  case (it.dir) of
  DIR_DOWN:
    (* Запись родителя в стек *)
    if (n > 99) then msg:='CheckValid: Stack overflow'; {goto __error} end_if;
    stack[n] := it.item;
    n:=n+1;
  DIR_UP:
    (* Извлечение из стека *)
    if (is_poly(it.item)) then  (* элемент - родитель *)
    
      (* Выборка потомства из стека *)
      m:=0;
      while (stack[n-1]<>it.item) do
        n:=n-1;
        if (m > 15) then msg:='CheckValid: Kids overflow'; {goto __error} end_if;
        kids[m]:=stack[n];
        m:=m+1;
      end_while;
      
      (* Анализ потомства *)
      for im:=0 to m-1 do
        PIT:=kids[im]; (* Позиция ребёнка *)
        msg:=MakeMsg('CheckValid: P=', ID2Str(IT_ID(IT.ITEM)), ', C=', ID2Str(IT_ID(PIT)));
        
        (* === Проверка 1: Если родитель в цилиндрической СК, то дети - тоже  *)
        if (is_cyl(IT.ITEM) and not is_cyl(PIT)) then
          msg := MakeMsg(msg, ', Er=CS does not match');
          { goto __exit;  }
        end_if;
        
        (* === Проверка 2: Размер не может быть нулевым  *)
        Sh := get_sh(PIT);
        P0 := sh.p0; (* Начало отсчёта  (абс) *)
        P1 := sh.pl; (* Начало элемента (лок) *)
        P2 := sh.lx; (* Размер элемента (лок) *)
        
        msg := MakeMsg(msg, ' LWH=(',REAL_TO_STRING(P2[0]), ','  );
        msg := MakeMsg(msg, '',      REAL_TO_STRING(P2[1]), ','  );
        msg := MakeMsg(msg, '',      REAL_TO_STRING(P2[2]), ');' );
        
        if (p2[0]<=0.1 or p2[1]<=0.1 or p2[2]<=0.1) then 
          msg := MakeMsg(msg, ', Er=LWH must be nonzero'); 
          {goto __exit} 
        end_if;

        (* Преобразуем точки p1, p2 в абсолютные координаты *)
        p2 := _point((p1[0]+p2[0]), (p1[1]+p2[1]), (p1[2]+p2[2]));
        
        p1 := Sh_Loc2Abs(Sh, p1[0], p1[1], p1[2]);
        p2 := Sh_Loc2Abs(Sh, p2[0], p2[1], p2[2]);
        
        msg := MakeMsg(msg, ' P1=(', REAL_TO_STRING(P1[0]), ','  );
        msg := MakeMsg(msg, '',      REAL_TO_STRING(P1[1]), ','  );
        msg := MakeMsg(msg, '',      REAL_TO_STRING(P1[2]), ');' );
        msg := MakeMsg(msg, ' P2=(', REAL_TO_STRING(P2[0]), ','  );
        msg := MakeMsg(msg, '',      REAL_TO_STRING(P2[1]), ','  );
        msg := MakeMsg(msg, '',      REAL_TO_STRING(P2[2]), ');' );
                        
        (* === Проверка 3: Точки p1, p2 элемента не могут быть вне родителя   *)
        Chk := Sh_Point2Dot(get_sh(IT.ITEM), p1[0], p1[1], p1[2]);
        if (Chk.V <= 0) then 
          msg := MakeMsg(msg, ', Er=P1 out of parent' ); 
          {goto __exit} 
        end_if;
        Chk := Sh_Point2Dot(get_sh(IT.ITEM), p2[0], p2[1], p2[2]);
        if (Chk.V <= 0) then 
          msg := MakeMsg(msg, ', Er=P2 out of parent' ); 
          {goto __exit} 
        end_if;

        (* === Проверка 4,5: *)
        if (not is_poly(PIT)) then
          for j:=0 to m-1 do
            (* Проверка 4: p1,p2 одного элемента не могут быть внутри другого *)
            if (j<>im) then
              PIT2:=kids[j];
              Chk := Sh_Point2Dot(get_sh(PIT2), p1[0], p1[1], p1[2]);
              if (Chk.V = 16#01 or Chk.V = 16#ff) then 
                msg := MakeMsg(msg, ', Err: P1 of ', SINT_TO_STRING(PIT));
                msg := MakeMsg(msg, ' is into ',   SINT_TO_STRING(PIT2));
                {goto __exit} 
              end_if;
              Chk := Sh_Point2Dot(get_sh(PIT2), p2[0], p2[1], p2[2]);
              if (Chk.V = 16#01 or Chk.V = 16#ff) then 
                msg := MakeMsg(msg, ', Err: P2 of ', SINT_TO_STRING(PIT));
                msg := MakeMsg(msg, ' is into ',   SINT_TO_STRING(PIT2));
                {goto __exit} 
              end_if;
            end_if;
            
            (* Проверка 5: *)
            (* --- *)
            
          end_for;
        end_if;
        
        msg:=LogMsg(msg);      
      end_for;
      
    else (* конечный элемент *)
      (* Запись конечного элемента в стек *)
      if (n > 99) then msg := 'CheckValid: Stack overflow'; {goto __error} end_if;
      stack[n] := it.item;
      n:=n+1;
    end_if;
    
  end_case;
  
  it := it_next(it);
end_while;

bRes:=true;

{ __exit: }
msg:=LogMsg(msg);
Do_CheckValid := bRes;
return;

{ __error: }
Do_CheckValid := st_set_stat(E_CHECKVALID, IT_ID(it.item), msg);

          
END_FUNCTION

(* Значение поля 'p' структуры var *)
FUNCTION var_d : TDot
  VAR_INPUT
    TV : TVar := 0;  (* Структура типа TVar *)
  END_VAR

            {{
  #pragma pack(push, 4)
  typedef union {
    TVAR tv;
    struct { USINT R:1;   INT A:15; USINT C:1;   INT B:15; };
    struct { USINT r:1; USINT d:2;   SINT p:8; USINT i:7; USINT j:7; USINT k:7; };
  } var_t, *pvar_t;
  #pragma pack(pop)

  // Величина должна быть ссылкой
  // ASSERT(1, NULL, pvar->r, TERROR__E_FAIL, __INIT_STRING);
  VAR_D.A.table[0] = ((pvar_t) &TV)->i;
  VAR_D.A.table[1] = ((pvar_t) &TV)->j;
  VAR_D.A.table[2] = ((pvar_t) &TV)->k;
  VAR_D.V          = ((pvar_t) &TV)->p;
}}

          
END_FUNCTION

(* Значение поля 'p' структуры var *)
FUNCTION var_p : TPos8
  VAR_INPUT
    TV : TVar := 0;  (* Структура типа TVar *)
  END_VAR

            {{
  #pragma pack(push, 4)
  typedef union {
    TVAR tv;
    struct { USINT R:1;   INT A:15; USINT C:1;   INT B:15; };
    struct { USINT r:1; USINT d:2;   SINT p:8; USINT i:7; USINT j:7; USINT k:7; };
  } var_t, *pvar_t;
  #pragma pack(pop)
  pvar_t pvar = (pvar_t)&TV;
  
  // Величина должна быть ссылкой
  // ASSERT(1, NULL, pvar->r, TERROR__E_FAIL, __INIT_STRING);
  VAR_P = pvar->p;
}}

          
END_FUNCTION

(* Установка флага деблокировки *)
FUNCTION st_set_ready : BOOL
  VAR_INPUT
    RDY : BOOL := FALSE;  (* Флаг деблокировки *)
  END_VAR

            {{ return (ST_SET_READY=(__GET_GLOBAL_STAT()->RDY=RDY)); }}

          
END_FUNCTION

(* Установка флага отладки *)
FUNCTION st_set_debug : BOOL
  VAR_INPUT
    DBG : BOOL := FALSE;  (* Флаг отладки *)
  END_VAR

            {{ return (ST_SET_DEBUG=(__GET_GLOBAL_STAT()->DBG=DBG)); }}

          
END_FUNCTION

(* Проверка флага деблокировки *)
FUNCTION st_is_ready : BOOL
  VAR_INPUT
    tmp : BOOL := FALSE;  (* Пустышка *)
  END_VAR

            {{ return (ST_IS_READY=__GET_GLOBAL_STAT()->RDY); }}

          
END_FUNCTION

(* Проверка флага отладки *)
FUNCTION st_is_debug : BOOL
  VAR_INPUT
    tmp : BOOL := FALSE;
  END_VAR

            {{ return (ST_IS_DEBUG=__GET_GLOBAL_STAT()->DBG); }}

          
END_FUNCTION

(* Информация по элементу *)
FUNCTION IT_InfoStr : STRING
  VAR_INPUT
    PIT : TPos8 := -1;  (* Позиция элемента *)
  END_VAR
  VAR
    Item : TItem;  (* Копия элемента *)
    Shape : TShape;  (* Геометрия элемента *)
    msg : STRING := '';  (* Строка информации *)
  END_VAR

            Item  := get_it(it_pos(PIT));
Shape := get_sh(PIT);
msg  := MakeMsg(msg, ' [',   ID2Str(Item.ID) );
msg  := MakeMsg(msg, ', P=', SINT_TO_STRING(Item.Par) );
msg  := MakeMsg(msg, ', O=(',REAL_TO_STRING(Shape.p0[0]), '');
msg  := MakeMsg(msg, ', ',   REAL_TO_STRING(Shape.p0[1]), '');
msg  := MakeMsg(msg, ', ',   REAL_TO_STRING(Shape.p0[2]), ')');
msg  := MakeMsg(msg, ', N=(',REAL_TO_STRING(Shape.pL[0]), '');
msg  := MakeMsg(msg, ', ',   REAL_TO_STRING(Shape.pL[1]), '');
msg  := MakeMsg(msg, ', ',   REAL_TO_STRING(Shape.pL[2]), ')');
msg  := MakeMsg(msg, ', W=(',REAL_TO_STRING(Shape.Lx[0]), '');
msg  := MakeMsg(msg, ', ',   REAL_TO_STRING(Shape.Lx[1]), '');
msg  := MakeMsg(msg, ', ',   REAL_TO_STRING(Shape.Lx[2]), ')]');
IT_InfoStr:=MSG;

          
END_FUNCTION

(* ГУ-2,3. Левые прогоночные коэффициенты *)
FUNCTION Alfa_03 : P_RERE
  VAR_INPUT
    Ht : REAL := 0.0;  (* Шаг по времени *)
    M : TMatter;  (* Свойства материи (a, l, h, k) *)
    Tn_0 : REAL := 0.0;  (* Тi левой границы (i=0) на пред шаге (t=n) *)
    Tq_0 : REAL := 0.0;  (* T среды Ti или поток qi (i=0) *)
    Qn_0 : REAL := 0.0;  (* Тепловыделение Qi (i=0) на пред шаге (t=n) *)
    V_0 : REAL := 0.0;  (* Скорость течения Vi (i=0) *)
    R_0 : REAL := 0.0;  (* Радиус дуги Ri (i=0) *)
    Bound3 : BOOL := TRUE;  (* Признак - краевое условие 3-го рода (по умолчанию) *)
  END_VAR
  VAR
    D_0 : REAL := 0.0;  (* Коэффициент Di (i=0) *)
    E_0 : REAL := 0.0;  (* Коэффициент Ei (i=0) *)
    b_0 : REAL := 0.0;  (* Коэффициент bi (i=0) *)
    k_0 : REAL := 0.0;  (* Коэффициент ki (i=0) *)
    h2 : REAL := 0.0;  (* Вспомогательная *)
    at2 : REAL := 0.0;  (* Вспомогательная *)
    DE : REAL := 0.0;  (* Вспомогательная *)
    denom : REAL := 0.0;  (* Знаменатель *)
    Res : P_RERE;  (* Пара - (A=alfa0, B=beta0) *)
  END_VAR

            if (R_0 > 1.0E-5) then 
  if (not Bound3) then M.k := 1.0; end_if;
  b_0 := M.k/M.l;
  k_0 := b_0*Tq_0;
  if (not Bound3) then b_0 := 0.0; end_if;
  if (R_0 < 1.0E5) then E_0 := M.h / (2.0*R_0); end_if;
  D_0 := (abs(V_0)*M.h) / (2.0*M.a);
else
  (* Малый радиус - условия симметрии h=0 *)
  M.h := 0.0;
end_if;

h2    := M.h * M.h;
at2   := 2.0 * M.a * Ht;
DE    := (1.0 + D_0 - E_0);
denom := h2 + at2 * (1.0 + DE * M.h*b_0);

Alfa_03.A := at2 / denom;
Alfa_03.B := ( h2 * (Tn_0 + Ht*Qn_0) + at2 * DE * M.h*k_0 ) / denom;
          
END_FUNCTION

(* ГУ-4. Левые прогоночные (A=alfa0, B=beta0) *)
FUNCTION Alfa_04 : P_RERE
  VAR_INPUT
    Ht : REAL := 0.0;  (* Шаг по времени *)
    M1 : TMatter;  (* Свойства материи-1 (a, l, h, k) *)
    M2 : TMatter;  (* Свойства материи-2 (a, l, h, k) *)
    Alfa : P_RERE;  (* Пара - A=alfa(0-1), B=beta(0-1) *)
    Tn_0 : REAL := 0.0;  (* Тi левой границы (i=0) на пред шаге *)
    Q1n_0 : REAL := 0.0;  (* Тепловыделение 1 *)
    Q2n_0 : REAL := 0.0;  (* Тепловыделение 2 *)
  END_VAR
  VAR
    A : REAL := 0.0;  (* Коэффициент A *)
    B : REAL := 0.0;  (* Коэффициент B *)
    F : REAL := 0.0;  (* Коэффициент F *)
  END_VAR

            (* Малый шаг - условие симметрии *)
if (M1.h < 1.0E-4 or M2.h < 1.0E-4) then
  Alfa_04.A := 1.0;
  Alfa_04.B := 0.0;
else
  (* Вариант-1: считаем известной T в точке i=-1, тогда Alfa.A=0, Alfa.B=T *)
  (* Вариант-2: считаем известной пару Alfa|Beta в точке i=-1 на момент расчёта *)

  A :=    M1.l / M1.h;

  B :=    (M1.l / M1.h) 
        + (M2.l / M2.h) 
        + (M1.l*M1.h/(2.0*M1.a*Ht))  
        + (M2.l*M2.h/(2.0*M2.a*Ht))
        - (M2.l / M2.h) * Alfa.A; (* Доп слагаемое - вариант 1 или 2 *)

  F :=  - Tn_0 * ( (M1.l*M1.h/(2.0*M1.a*Ht)) + (M2.l*M2.h/(2.0*M2.a*Ht)) ) 
        - (M1.l*M1.h/(2.0*M1.a)) * Q1n_0  
        - (M2.l*M2.h/(2.0*M2.a)) * Q2n_0 
        - (M2.l / M2.h) * Alfa.B; (* Доп слагаемое - вариант 1 или 2 *)

  Alfa_04.A :=  A/B;
  Alfa_04.B := -F/B;
end_if;
          
END_FUNCTION

(* Прогоночные коэффициенты i узла *)
FUNCTION Alfa_i : P_RERE
  VAR_INPUT
    Ht : REAL := 0.0;  (* Шаг по времени *)
    M : TMatter;  (* Свойства материи (a, l, h, k) *)
    Alfa_im : P_RERE;  (* Пара - alfa(i-1), B=beta(i-1) *)
    Ti : REAL := 0.0;  (* Тi на пред шаге *)
    Qi : REAL := 0.0;  (* Тепловыделение Qi (i=0) *)
    Vi : REAL := 0.0;  (* Скорость течения Vi (i=0) *)
    Ri : REAL := 0.0;  (* Радиус дуги Ri (i=0) *)
  END_VAR
  VAR
    Ai : REAL := 0.0;  (* Коэффициент Ai *)
    Bi : REAL := 0.0;  (* Коэффициент Bi *)
    Ci : REAL := 0.0;  (* Коэффициент Ci *)
    Fi : REAL := 0.0;  (* Коэффициент Fi *)
    rh : REAL := 0.0;  (* Отношение rh=dt/h *)
    rk : REAL := 0.0;  (* Число Куранта rk=(a*dt)/h*h *)
    Via : REAL := 0.0;  (* Via = abs(Vi) *)
    Vip : REAL := 0.0;  (* Vip = Vi+ = (abs(Vi)+Vi)/2 *)
    Vim : REAL := 0.0;  (* Vim = Vi- = (abs(Vi)-Vi)/2 *)
    Di : REAL := 0.0;  (* Di = (Via * h ) / (2 * a) *)
    Ei : REAL := 0.0;  (* Ei = h / (2 *Ri) *)
    denom : REAL := 0.0;  (* Знаменатель *)
  END_VAR

            (* Малый радиус - условие симметрии *)
if (Ri < 1.0E-4) then 
  Alfa_i.A := 1.0;
  Alfa_i.B := 0.0;
else

  (* расчёт движения по радиусу *)
  if (Ri < 1.0e5) then Ei := M.h / (2.0 * Ri); end_if;
  
  (* расчёт движения среды *)
  if (Vi <> 0.0) then
    Via := abs(Vi);
    Vip := (Via + Vi)   / 2.0;
    Vim := (Via - Vi)   / 2.0;
    Di  := (Via * M.h)  / (2.0 * M.a);
  end_if;

  rh := Ht / M.h;       (* Отношение     (rh=dt/dx)     *)
  rk := (M.a*rh) / M.h; (* Число Куранта (rk=a*dt/dx^2) *)

  Ai :=       rk*(1.0+Ei) / (1.0+Di) + Vim*rh; 
  Ci :=       rk*(1.0-Ei) / (1.0+Di) + Vip*rh; 
  Bi := 1.0 +    (2.0*rk) / (1.0+Di) + Via*rh; 
  Fi := -Ti - Ht*Qi;

  denom := (Bi - Ci*Alfa_im.A);

  Alfa_i.A := Ai / denom;
  Alfa_i.B := (Ci*Alfa_im.B - Fi) / denom;
end_if;

          
END_FUNCTION

(* ГУ-2,3. Правая температура T(N) *)
FUNCTION Beta_N3 : REAL
  VAR_INPUT
    Ht : REAL := 0.0;  (* Шаг по времени *)
    M : TMatter;  (* Свойства материи (a, l, h, k) *)
    Alfa_N1 : P_RERE;  (* Пара - A=alfa(N-1), B=beta(N-1) *)
    Tn_N : REAL := 0.0;  (* Т правой границы (i=N) на пред t-шаге (t=n) *)
    Tq_N : REAL := 0.0;  (* T среды Ti или поток qi (i=N) *)
    Qn_N : REAL := 0.0;  (* Тепловыделение Qi (i=N) на пред t-шаге (t=n) *)
    V_N : REAL := 0.0;  (* Скорость течения Vi (i=N) *)
    R_N : REAL := 0.0;  (* Радиус дуги Ri (i=N) *)
    Bound3 : BOOL := TRUE;  (* Признак - краевое условие 3-го рода (по умолчанию) *)
  END_VAR
  VAR
    D_N : REAL := 0.0;  (* Коэффициент Di (i=N) *)
    E_N : REAL := 0.0;  (* Коэффициент Ei (i=N) *)
    b_N : REAL := 0.0;  (* Коэффициент bi (i=N) *)
    k_N : REAL := 0.0;  (* Коэффициент ki (i=N) *)
    h2 : REAL := 0.0;  (* Вспомогательная *)
    at2 : REAL := 0.0;  (* Вспомогательная *)
    DE : REAL := 0.0;  (* Вспомогательная *)
    denom : REAL := 0.0;  (* Знаменатель *)
  END_VAR

            if (R_N > 1.0E-5) then 
  if (not Bound3) then M.k := 1.0; end_if;
  b_N := M.k/M.l;
  k_N := b_N*Tq_N;
  if (not Bound3) then b_N := 0.0; end_if;
  if (R_N < 1.0E5) then E_N := M.h / (2.0*R_N); end_if;
  D_N := (abs(V_N)*M.h) / (2.0*M.a);
else
  (* Малый радиус - условия симметрии h=0 *)
  M.h := 0.0;
end_if;

h2    := M.h * M.h;
at2   := 2.0 * M.a * Ht;
DE    := (1.0 - D_N + E_N);
denom := h2 + at2 * (1.0 + DE * M.h*b_N - Alfa_N1.A);

Beta_N3 := ( h2 * (Tn_N + Ht*Qn_N) + at2 * (Alfa_N1.B + DE * M.h*k_N) ) / denom;

          
END_FUNCTION

(* ГУ-4. Правая температура T(N) *)
FUNCTION Beta_N4 : REAL
  VAR_INPUT
    Ht : REAL := 0.0;  (* Шаг по времени *)
    M1 : TMatter;  (* Свойства материи 1 *)
    M2 : TMatter;  (* Свойства материи 2 *)
    Alfa_Nm1 : P_RERE;  (* Пара - A=alfa(N-1), B=beta(N-1) *)
    Tn_N : REAL := 0.0;  (* Тi правой границы (i=N) на пред шаге *)
    Tn_Np1 : REAL;  (* Температура в точке (N+1) *)
    Q1n_N : REAL := 0.0;  (* Тепловыделение 1 *)
    Q2n_N : REAL := 0.0;  (* Тепловыделение 2 *)
  END_VAR
  VAR
    B : REAL := 0.0;  (* Коэффициент B *)
    C : REAL := 0.0;  (* Коэффициент C *)
    F : REAL := 0.0;  (* Коэффициент F *)
  END_VAR

            (* Малый шаг - условие симметрии *)
if (M1.h < 1.0E-4 or M2.h < 1.0E-4) then
  Beta_N4 := Tn_Np1;
else
  (* Cчитаем известной T=Tn_Np1 в точке i=N+1, тогда Alfa.A=0, Alfa.B=T *)
  C :=  M1.l / M1.h;

  B :=    (M1.l / M1.h) 
        + (M2.l / M2.h) 
        + (M1.l * M1.h / (2.0*M1.a*Ht))  
        + (M2.l * M2.h / (2.0*M2.a*Ht));

  F :=  - Tn_N * ( (M1.l*M1.h/(2.0*M1.a*Ht)) + (M2.l*M2.h/(2.0*M2.a*Ht)) ) 
        - (M1.l * M1.h / (2.0*M1.a)) * Q1n_N  
        - (M2.l * M2.h / (2.0*M2.a)) * Q2n_N
        - (M2.l / M2.h) * Tn_Np1; (* доп слагаемое - см. Tn_Np1 *)

  Beta_N4 := (C * Alfa_Nm1.B - F) / (B - C * Alfa_Nm1.A);
end_if;
          
END_FUNCTION

(* Коэффициент теплоотдачи воздуха *)
FUNCTION kto_air : REAL
  VAR_INPUT
    L : REAL := 0.0;  (* Определяющий размер *)
  END_VAR

            kto_air:=10.0;
          
END_FUNCTION

(* Коэффициент теплоотдачи масла *)
FUNCTION kto_oil : REAL
  VAR_INPUT
    L : REAL := 0.0;  (* Эквивалентный диаметр *)
    dTm : REAL := 0.0;  (* Перепад температуры масло - поверхность *)
  END_VAR
  VAR CONSTANT
    C : REAL := 0.59;  (* Эмпирическая константа *)
    n : REAL := 0.25;  (* Эмпирическая константа *)
  END_VAR

            kto_oil:=36.0;
          
END_FUNCTION

(* Обратная прогонка *)
FUNCTION Temp_i : REAL
  VAR_INPUT
    _Alfa_i : P_RERE;  (* Пара - alfa(i+1), B=beta(i+1) *)
    T_ip : REAL := 0.0;  (* Температура предыдущего узла *)
  END_VAR

            Temp_i := _Alfa_i.A * T_ip + _Alfa_i.B;

          
END_FUNCTION

(* Сборка материи *)
FUNCTION _Matter : TMatter
  VAR_INPUT
    a : REAL := 0.0;  (* Параметр h *)
    l : REAL := 0.0;  (* Параметр l *)
    h : REAL := 0.0;  (* Параметр h *)
    k : REAL := 0.0;  (* Параметр k *)
  END_VAR

            _Matter.a:=a;
_Matter.l:=l;
_Matter.h:=h;
_Matter.k:=k;

          
END_FUNCTION

(* Расчёт элемента по направлению Ix *)
FUNCTION IT_Process : TError
  VAR_INPUT
    PIT : TPos8 := -1;  (* Позиция элемента *)
    Ix : USINT := 0;  (* Индекс направления (0-Ox,1-Oy,2-Oz) *)
    CDT : DT := DT#2000-01-01-00:00:00;  (* Текущее время расчёта *)
  END_VAR
  VAR
    PDT : DT := DT#2000-01-01-00:00:00;  (* Предыдущее время расчёта *)
    It : TItem;  (* Элемент расчёта *)
    Hd : THead;  (* Заголовок модели *)
    Sh : TShape;  (* Фигура элемента *)
    Ax : USINT := 0;  (* Направление оси *)
    Ox : TAxO;  (* Индексы внешних координат *)
    Cx : TAxO;  (* Порядок перебора координат *)
    Q : SINT := 0;  (* Номер квадранта i-узла *)
    Ht : REAL := 0.0;  (* Шаг по времени (сек) *)
    K : ARRAY[0..2] OF INT;  (* Индексы циклов перебора X,Y,Z *)
    L : ARRAY[0..2] OF INT;  (* Граница, координата X,Y,Z *)
    H0 : TPoint := [0.0, 0.0, 0.0];  (* Шаги по координатам-1 (оригинал) *)
    Hx2 : TPoint := [0.0, 0.0, 0.0];  (* Смещение по координатам-2 *)
    pR : TPoint := [0.0, 0.0, 0.0];  (* Конечная точка *)
    Iv : SINT := 0;  (* Индекс связанной величины-1 *)
    Im : SINT := 0;  (* Индекс материала-1 (свой) *)
    V : TVal;  (* Cвязанная величина *)
    Vx : REAL := 0.0;  (* Значение связанной величины-1 *)
    Px : TProf;  (* Профиль связанной величины-1 (своей) *)
    Cm : TMat;  (* Материал элемента-1 *)
    Pm : TProps;  (* Свойства материала-1 *)
    P0 : TPoint := [0.0, 0.0, 0.0];  (* Точка начала нити (абс) *)
    Hi : REAL := 0.0;  (* Шаг по координате *)
    Hi2 : REAL := 0.0;  (* Шаг по координате-2 *)
    Pi : TPoint := [0.0, 0.0, 0.0];  (* Точка i-узла нити (лок) *)
    Ri : REAL := 0.0;  (* Радиус дуги в узле i элемента-1 *)
    Li : REAL := 0.0;  (* Левая граница по Ix *)
    Vi1 : REAL := 0.0;  (* Скорость движения в узле i элемента-1 *)
    Qi1 : REAL := 0.0;  (* Тепловыделение в узле i элемента-1 *)
    Ti1 : REAL := 0.0;  (* Температура в узле i элемента-1 *)
    M : TMatter;  (* Свойства материи-1 *)
    P : TPoint := [0.0, 0.0, 0.0];  (* Вспомогательная точка *)
    TV : TVar := 0;  (* Вспомогательная точка *)
    LR : ARRAY[0..3] OF P_BOOL := [FALSE, FALSE, FALSE, FALSE];  (* Флаги формы границ по радиусу *)
    PIT2 : TPos8 := -1;  (* Позиция элемента-2 *)
    Kn2 : TKnot := [0, 0, 0];  (* Количество узлов сетки-2 *)
    Im2 : SINT := 0;  (* Индекс материала-2 *)
    Cm2 : TMat;  (* Материал элемента-2 *)
    Pm2 : TProps;  (* Свойства материала-2 *)
    Iv2 : SINT := 0;  (* Индекс связанной величины-2 *)
    V2 : TVal;  (* Cвязанная величина-2 *)
    Vx2 : REAL := 0.0;  (* Значение связанной величины-2 *)
    Px2 : TProf;  (* Профиль связанной величины-2 *)
    Vi2 : REAL := 0.0;  (* Скорость движения в узле i элемента-2 *)
    Qi2 : REAL := 0.0;  (* Тепловыделение в узле i элемента-2 *)
    Ti2 : REAL := 0.0;  (* Температура в узле i элемента-2 *)
    M2 : TMatter;  (* Свойства материи элемента-2 *)
    Tmid2 : REAL := 0.0;  (* Средняя температура элемента-2 *)
    i : INT := 0;  (* Индекс расчётной нити *)
    N : INT := 0;  (* Правый предел расчётной нити *)
    off : P_INT;  (* Cмещение и размер ячейки *)
    xx : REAL := 0.0;  (* Вспомогательная переменная *)
    ii : INT := 0;  (* Вспомогательная переменная *)
    Alfa : P_RERE;  (* Пара - A=alfa(N-1), B=beta(N-1) *)
    Alfas : ARRAY[0..63] OF P_RERE;  (* Коэффициенты прогонки alfa, beta *)
    iRes : TError := E_SUCCESS;  (* Результат выполнения *)
    bRes : BOOL := false;  (* Результат выполнения *)
    msg : STRING := '';  (* Строка в протокол *)
  END_VAR
  VAR CONSTANT
    Kt : REAL := 300.0;  (* Масштаб по времени (кратность) *)
    Hmin : REAL := 1.0E-5;  (* Минимальный шаг по координате *)
  END_VAR

            (* Получаем время предыдущего расчёта и сохраняем текущее *)
PDT := get_pdt(PIT, Ix);
PIT := set_pdt(PIT, Ix, CDT);

Hd := get_h(0);       (* Заголовок модели *)
It := get_it(PIT);    (* Элемент          *)
Sh := get_sh(PIT);    (* Фигура элемента  *)
Ax := sh_get_ax(Sh);  (* Направление оси  *)

Im := It.Im;          (* Индекс материала *)
Iv := It.Iv;          (* Индекс величины  *)

Cm := get_mt(It.Im);  (* Материал *)

(* Получение значения динамической величины элемента-1 и её профиля *)
if (Iv > 0 and Iv < Hd.Nv) then
  V  := get_vl(It.Iv);
  Vx := get_bf(V.Iv) * sint_to_real(V.Vi[Ix].A);
  Px := get_pr(V.Vi[Ix].B);
end_if;

(* Ориентация элемента *)
Ox := AXO(Ax,  TRUE);     (* Порядок перебора координат *)
Cx := AXO(Ix+1, FALSE);   (* Порядок обхода сетки       *)

(* Признаки материала *)
Pm.Air   := (Im = 0);            (* Признак - воздух (нулевой материал) *)
Pm.Oil   := (Cm.MD <> 0.0);      (* Признак - масло  (задана вязкость)  *)
Pm.Fluid := (Pm.Oil or Pm.Air);  (* Признак - флюид  (воздух или масло) *)
Pm.Solid := (not Pm.Fluid);      (* Признак - твердое тело (не флюид)   *)

(* Если элемент - воздух - не считаем *)
if (Pm.Air) then {goto __exit} end_if;

(* Опредедение шага (Ht>0) по времени в секундах *)
Ht := 300.0; (*Kt * ULINT_TO_REAL(DT_TO_ULINT(CDT)-DT_TO_ULINT(PDT));*)
if (Ht < 1.0) then iRes:=E_TIMESIZE; {goto __exit} end_if;

(* Опредедение шага по сетке (ориг) *)
H0 := _point( Sh.Lx[0]/INT_TO_REAL(Sh.Kn[0]-1), 
              Sh.Lx[1]/INT_TO_REAL(Sh.Kn[1]-1), 
              Sh.Lx[2]/INT_TO_REAL(Sh.Kn[2]-1) );
if ( (H0[0]<Hmin) or (H0[1]<Hmin) or (H0[2]<Hmin) ) 
  then iRes:=E_STEPSIZE; {goto __exit} end_if;

(* TEST *)
(* Имитация тепловыделения в обмотках низкого и высокого напряжения *)
if (PIT = 21 or PIT = 31) then Vx := 5.0; end_if;
if (PIT = 38 or PIT = 59 or PIT = 80) then Vx := 3.0;  end_if;
if (PIT = 42 or PIT = 63 or PIT = 84) then Vx := 12.0; end_if;
if (PIT = 45 or PIT = 46 or PIT = 47 or PIT = 48 or PIT = 49 or 
    PIT = 50 or PIT = 51 or PIT = 52 or PIT = 53 or PIT = 54) then Vx := 20.0; end_if;
if (PIT = 66 or PIT = 67 or PIT = 68 or PIT = 69 or PIT = 70 or 
    PIT = 71 or PIT = 72 or PIT = 73 or PIT = 74 or PIT = 75) then Vx := 20.0; end_if;
if (PIT = 87 or PIT = 88 or PIT = 89 or PIT = 90 or PIT = 91 or 
    PIT = 92 or PIT = 93 or PIT = 94 or PIT = 95 or PIT = 96) then Vx := 20.0; end_if;

(* Базовые значения профилируемых величин-1 - "равномерно без профиля" *)
if (Vx=0.0) then Vi1 := 0.0; Qi1 := 0.0;
else
  if (Pm.Fluid) then Vi1 := abs(Vx);                    (* скорость       *)
  else Qi1 := Vx/INT_TO_REAL(Sh.Kn[0]*Sh.Kn[1]*Sh.Kn[2]);  (* тепловыделение *)
  end_if; 
end_if;

(* Сохранение верхних индексов узлов сетки по координатным осям *)
L[Cx.x] := Sh.Kn[0]-1; (* =2 при iX=0 *)
L[Cx.y] := Sh.Kn[1]-1; (* =0 при iX=0 *)
L[Cx.z] := Sh.Kn[2]-1; (* =1 при iX=0 *)
N:=L[2];  (* верхний индекс прогонки *)

(* Циклы по сетке в направлении Ix *)
K[0]:=0;
while (K[0] <= L[0]) do (* Цикл (0) *)
  K[1]:=0;
  while (K[1] <= L[1]) do (* Цикл (1) *)
    K[2]:=0;
  
    (* Локальная точка элемента в начале нити *)
    P0 := _point( Sh.pL[0] + H0[0]*INT_TO_REAL(K[Cx.x]), 
                  Sh.pL[1] + H0[1]*INT_TO_REAL(K[Cx.y]),
                  Sh.pL[2] + H0[2]*INT_TO_REAL(K[Cx.z]) );

    (* Коррекция начальной точки и шага в направлении радиуса *)
    if (Ax<>0 (*and Ix=Ox.x*)) then
      P0[Ox.y] := angle(P0[Ox.y], Sh.pL[Ox.y]);
      P := Reform(Sh.wF, P0[Ox.y], P0[Ox.x], Sh.pL[Ox.x], Sh.Lx[Ox.x]);
      P0[Ox.x] := P[0];                 (* коррекция начальной точки *)
      H0[Ox.x] := P[2]/INT_TO_REAL(N);  (* коррекция шага по радиусу *)
    end_if;
                                                      
    (* === Прямая прогонка === *)
    for i:=0 to N do (* Цикл (2) - прогонка по направлению Ix *)
      K[2]   := i;                      (* i -  индекс нити прогонки *)
      Pi     := P0;                     (* P0 - начальная точка нити *)
      Pi[Ix] := P0[Ix] + 
                H0[Ix]*INT_TO_REAL(i);  (* текущая точка узла        *)
      
      (* Расчёт радиуса Ri и шага Hi *)
      if (Ax<>0 and Ix=Ox.x) then    (* движение по радиусу       *)
        Ri := Pi[Ix]   * 0.001;         (* мм->м                     *)
        Hi := H0[Ix]   * 0.001;         (* мм->м                     *)
      elsif (Ax<>0 and Ix=Ox.y) then (* движение по дуге          *)
        P  := Reform(Sh.wF, Pi[Ox.y], Pi[Ox.x], Sh.pL[Ox.x], Sh.Lx[Ox.x]);
        Pi[Ox.x] := P[0];               (* радиальная координата     *)
        Ri := Pi[Ox.x] * 0.001;         (* мм->м                     *)
        Hi := Ri * radi(H0[Ix]);        (* длина дуги (м)            *)
      else                              (* "плоское" движение        *)
        Ri := 1.0e6;                    (* большой радиус            *)
        Hi := H0[Ix]   * 0.001;         (* мм->м                     *)
      end_if;

      (* Свойства материи M(a, lambda, h, k) *)
      M := _Matter(Cm.kt/(Cm.PL*Cm.CP), Cm.kt, Hi);
      
      (* Смещение расчётного узла в сетке *)
      Off := knoff(Sh.Kn[0], Sh.Kn[1], Sh.Kn[2], K[Cx.x], K[Cx.y], K[Cx.z]);
      
      (* Температура расчётного узла (код (int) -> °С (real)) *)
      Ti1 := C2T(var_v( get_var(its_gr(0), PIT, Off) )); 
      
      (* Обработка краевых условий *)
      if ((i = 0) or (i = N)) then
      
        (* Получение дескриптора смежного элемента (PIT2) *)
        TV   := get_var(its_gr(0), PIT, Off, Ix+1);
        PIT2 := var_p(TV); (* может быть = (-1) *)
        
        {{
          // Доступ к свойствам элемента-2
          TITEM *pItem2 = ((PIT2==-1) ? NULL : &(__GET_GLOBAL_ITS()->IT.table[PIT2]));
          IM2 = ((pItem2==NULL) ? 0 : pItem2->IM);  // Индекс материала
          CM2 = GET_MT(1,NULL,IM2);                 // Материал
          
          if (IM2==0) { // воздух =>
            VX2 = 0.0;                              // динимаческая величина = 0
          } else {      // обычный элемент =>
            IM2 = pItem2->IM;                       // Индекс материала
            IV2 = pItem2->IV;                       // Индекс величины

            __ARRAY_OF_TVAL_25  *pVAL = &__GET_GLOBAL_STS()->VL; // Связанные величины
            __ARRAY_OF_TPROF_30 *pPRO = &__GET_GLOBAL_STS()->PR; // Профили
            __ARRAY_OF_REAL_32  *pBUF = &__GET_GLOBAL_STS()->BF; // Буфер величин
                        
            if (IV2 > 0 && IV2 < HD.NV) {
              VX2 = pVAL->table[IV2].VI.table[IX].A * pBUF->table[pVAL->table[IV2].IV];
              PX2 = pPRO->table[pVAL->table[IV2].VI.table[IX].B];
            }
          }
          
        }}
        
        (*Kn2   := it_kn(PIT2);*) (* размерность сетки элемента-2 *)
        
        (* времяночка - заплатка *)
        Tmid2 := C2T(cn_mid(get_cn(PIT2)));
        
        (* Признаки материала 2 (соседа) *)
        Pm2.Air   := (Im2 = 0);             (* Признак - воздух (Im=0)         *)
        Pm2.Oil   := (Cm2.md <> 0.0);       (* Признак - масло  (md<>0)        *)
        Pm2.Fluid := (Pm2.Oil or Pm2.Air);  (* Признак - флюид  (Air or Oil)   *)
        Pm2.Solid := (not Pm2.Fluid);       (* Признак - твердое тело          *)

        (* Базовые значения профилируемых величин-2 - "равномерно без профиля" *)
        if (Vx2=0.0) then Vi2 := 0.0; Qi2 := 0.0;
        else
          if (Pm2.Fluid) then Vi2 := abs(Vx2);
          else Qi2 := Vx2/INT_TO_REAL( 4096 (*Kn2[0] * Kn2[1] * Kn2[2]*) ); 
          end_if; 
        end_if;

        (* Запрашиваем температуру в узле сетки-2, ближайшем к точке расчёта *)
        (*
        P   := Sh_Loc2Abs(PIT, Pi[0], Pi[1], Pi[2]);
        TV := IT_Check(PIT2, P[0], P[1], P[2], false);
        *)
        
        Ti2 := C2T(var_v(TV)); (* код (int) -> °С (real) *)
        
        (* TV.PT := Sh_Dot2Point(PIT2, var_d(TV.TV)) *)
        (* Hi2 := abs(P[Ix]-TV.PT[Ix]); *)
        
        (*+*)   if (K[0]=0 and K[1]=0 and PIT=3) then
                  msg := MakeMsg(   '-> Ti2= ', REAL_TO_STRING(Ti2));
                  msg := MakeMsg(msg, ' off= ', INT_TO_STRING(OFF.A));
                  msg := MakeMsg(msg, ' PIT= ', SINT_TO_STRING(PIT2));
                  msg := MakeMsg(msg, ' Hi2= ', REAL_TO_STRING(Hi2));
                  msg := LogMsg (msg);
                end_if; 
                                                
        (* Свойства материи-2 *)
        M2 := _Matter(Cm2.kt/(Cm2.PL*Cm2.CP), Cm2.KT, (* Hi2* *)0.001); (* в метрах *)
        
        (* === Метод прогонки === *)
        if (i = 0) then (* левая граница *)
        
          (* --- Расчёт коэффициентов Alfas[0] на левой границе --- *)
          if (Pm2.Air) then (* ГУ-3 *)
          
            if (true) then
              M.k := kto_air(1.0);
              Alfas[0] := Alfa_03(Ht, M, Ti1, Ti2, Qi1, Vi1, Ri);
            else
              Alfa.A := 0.0; Alfa.B := Ti2; 
              Alfas[0] := Alfa_i(Ht, M, Alfa, Ti1, Qi1, Vi1, Ri);
            end_if;
            
          elsif ((*(Pm.Oil and Pm2.Solid) or*) (Pm.Solid and Pm2.Oil)) then
          
              M.k := kto_oil(1.0);
              Alfas[0] := Alfa_03(Ht, M, Ti1, Tmid2-(Tmid2-20.0)/2.2, Qi1, Vi1, Ri);
          
          else  (* ГУ-4 *)
          
            Alfa.A := 0.0; Alfa.B := Ti2; 
            if (true) then
              (* Вариант 1 *)
              Alfas[0] := Alfa_i(Ht, M, Alfa, Ti1, Qi1, Vi1, Ri);
            else
              (* Вариант 2 *)
              M2.h := 0.001;
              Alfas[0] := Alfa_04(Ht, M, M2, Alfa, Ti1, Qi1, Qi2);
            end_if;
            
          end_if;
          
        elsif (i = N) then (* правая граница *)
        
          (* --- Расчёт температуры T[N] на правой границе --- *)
          if (Pm2.Air) then (* ГУ-3 *)
          
            if (true) then
              M.k := kto_air(1.0);
              xx := Beta_N3(Ht, M, Alfas[N-1], Ti1, Ti2, Qi1, Vi1, Ri);
            else
              Alfas[N] := Alfa_i(Ht, M, Alfas[N-1], Ti1, Qi1, Vi1, Ri);
              xx := Temp_i(Alfas[N], Ti2);
            end_if;
            
          elsif ((*(Pm.Oil and Pm2.Solid) or*) (Pm.Solid and Pm2.Oil)) then
          
              M.k := kto_oil(1.0);
              xx := Beta_N3(Ht, M, Alfas[N-1], Ti1, Tmid2-(Tmid2-20.0)/2.2, Qi1, Vi1, Ri);
          
          else (* ГУ-4 *)
          
            if (true) then
              (* Вариант 1 *)
              (*M.h := Hx2[Ix] * 0.001;*)
              Alfas[N] := Alfa_i(Ht, M, Alfas[N-1], Ti1, Qi1, Vi1, Ri);
              xx := Temp_i(Alfas[N], Ti2);
            else
              (* Вариант 2 *)
              M2.h := 0.001;
              xx := Beta_N4(Ht, M, M2, Alfas[N-1], Ti1, Ti2, Qi1, Qi2);
            end_if;
            
          end_if;
          
          (* Запись значения xx в сетку, °С (real) -> код (int) *)
          PIT := set_var(its_gr(0), PIT, OFF, _var(T2C(xx)));
          
          (*+*)     if (K[0]=0 and K[1]=0 and PIT =3) then
                      msg := MakeMsg(' T[', INT_TO_STRING(i), ']= ', REAL_TO_STRING(xx));
                      msg := MakeMsg(msg, ' M.a=', REAL_TO_STRING(M.a));
                      msg := MakeMsg(msg, ' M.h=', REAL_TO_STRING(M.h));
                      msg := MakeMsg(msg, ' M.l=', REAL_TO_STRING(M.l)); 
                      msg := MakeMsg(msg, ' R=',   REAL_TO_STRING(Ri));
                      msg := LogMsg(msg);
                    end_if; 
                    
        end_if;

      else (* не краевые точки *)
        (* --- Расчёт коэффициентов Alfas[i], Betas[i] --- *)
        Alfas[i] := Alfa_i(Ht, M, Alfas[i-1], Ti1, Qi1, Vi1, Ri);
      end_if; (* Обработка краевых условий *)

    end_for; (* прямая прогонка *)

    (* === Обратная прогонка === *)
    for i:=N-1 to 0 by -1 do
      K[2]:=i;
      
      (* --- Расчёт температуры T[N-1]..T[0] --- *)
      xx := Temp_i(Alfas[i], xx);
      
      (* Запись значения xx в сетку, °С (real) -> код (int) *)
      Off := knoff(Sh.Kn[0], Sh.Kn[1], Sh.Kn[2], K[Cx.x], K[Cx.y], K[Cx.z]);
      
      PIT := set_var(its_gr(0), PIT, Off, _var(T2C(xx)));
      
      (*+*) if (K[0]=0 and K[1]=0 and PIT =3) then
              msg := MakeMsg('T[', INT_TO_STRING(i), ']= ', REAL_TO_STRING(xx));
              msg := LogMsg(msg);
            end_if; 
            
    end_for; (* обратная прогонка *)
    
    K[1] := K[1]+1;
  end_while; (* Цикл (1) *)
  K[0] := K[0]+1;
end_while; (* Цикл (0) *)

{ __exit: }
IT_PROCESS := iRes;
          
END_FUNCTION

(* Процесс расчёта модели (обход дерева) *)
FUNCTION_BLOCK Process_XYZ
  VAR_EXTERNAL
    rTest : REAL;  (* Внешний буфер *)
    HDR : THead;  (* Внешний заголовок модели *)
    ITS : TItems;  (* Внешний массив элементов *)
  END_VAR
  VAR_INPUT
    IN : BOOL := TRUE;  (* Вход: Деблокировка *)
    Ix : USINT := 0;  (* Вход: Индекс направления расчёта *)
    N : SINT := -1;  (* Вход: N элементов, обрабатываемых за один вызов (-1= все) *)
  END_VAR
  VAR_OUTPUT
    bRes : BOOL := FALSE;  (* Выход: Результат расчёта (код ошибки) *)
  END_VAR
  VAR
    iErr : TError := E_SUCCESS;  (* Выход: Результат расчёта (код ошибки) *)
    i : SINT := 0;  (* Счётчик элементов, обрабатываемых за один вызов *)
    Ix_local : USINT := 0;  (* Индекс направления расчёта (локальная копия) *)
    bRestart : BOOL := true;  (* Флаг инициализации блока *)
    bBreak : BOOL := false;  (* Флаг выхода из цикла *)
    It : TIter;  (* Итератор дерева *)
    CDT : DT := DT#2000-01-01-00:00:00;  (* Текущее время расчёта *)
    PDT : DT := DT#2000-01-01-00:00:00;  (* Предыдущее время расчёта *)
    msg : STRING := '';  (* Строка протокола *)
    rr : REAL := 0.0;  (* Вспомогательная переменная *)
    RTIME : RTC;
    DTIME : TON;
  END_VAR

            IF (IN) THEN                          (* Деблокировка блока          *)
  IF (bReStart) THEN                  (* Инициализация блока         *)
    (* Проверка корректности конфигурации перед стартом *)
    if (Ix<0 or Ix>2) then iErr:=E_AXIS; {goto __error;} end_if;
    if (true) then
      (* Инициализация *)
      msg:=MakeMsg('== PROCESS init ... ');
      i:=0; it:=it_end(-1);
      bRes      := true;               
      bReStart  := false;
      bBreak    := false;
      Ix_local  := Ix;                 (* Направление запоминается    *)
      RTIME(EN  := false);             (* Текущее время -> PDT        *)
      RTIME(EN  := true, PDT := DT#2000-01-01-00:00:00, CDT => CDT);
      DTIME(IN  := false);             (* Рестарт счётчика DTIME      *)
      DTIME(IN  := true, PT := T#24h);
      PDT := CDT;
      (* Заносим время расчёта по направлению Ix в каждый элемент    *)
      it := it_begin(ID2PIT(0));
      while (it.item<>-1) do
        if (it.dir = DIR_UP) then ITS.IT[it.item].PDT[Ix]:=CDT; end_if;
        it := it_next(it);
      end_while;
      msg:=LogMsg(MakeMsg(msg, 'Ok! [time=', DT_TO_STRING(CDT),  '];'));
    end_if;
    RETURN; (* После инициализации - выход из блока *)
  END_IF;

  (* Проверка условий выполнения (нет ли блокировки на уровне модели) *)
  if (not st_is_ready(0)) then {goto __error;} end_if;
  (*bRes := TRUE;*)
  
  (* Проверка вхождения точки в модель *)
  (* TEST *) (*it := it_begin(42);*) 
  if (N<>0 and it.item=-1) then it := it_begin(ID2PIT(0)); end_if;

  (* TEST *) if (Ix_local=0) then msg:=LogMsg(MakeMsg(msg, 'START')); end_if;

  while (not bBreak and it.item<>-1) do
    case (it.dir) of
    DIR_UP:
      (* ВОПРОС: считаемем только конечные элементы? - пока да...  *)
      if (not is_poly(it.item)) then
        (* Крутим таймер - определяем текущее время расчёта *)
        DTIME(); 
        CDT := ULINT_TO_DT(ADD(DT_TO_ULINT(PDT), TIME_TO_ULINT(DTIME.ET)));
        
(* TEST -------- *)        
if (
  (it.item>=1 and it.item<=99) 
) then 
(* ------------- *)        
        (* === Расчёт элемента по направлению Ix === *)
        msg:=MakeMsg(msg, 'Process item ID=', ID2Str(IT_ID(it.item)), ' ... '); 
        
        iErr := IT_Process(it.item, Ix_local, CDT);
        bRes := (iErr = E_SUCCESS);
        if (not bRes) then 
          msg:=LogMsg(MakeMsg(msg, 'FAILED!'));
          {goto __error;} 
        else 
          msg:=LogMsg('');
        end_if;
(* ------------- *)        
end_if;        
(* ------------- *)        

      end_if; (* not is_poly(it.item) *)
    end_case; (* it.dir *)

    it := it_next(it);
    (* Проверка на досрочный выход из цикла *)
    if (not bBreak and N<>-1) then
      i:=i+1;
      if (i >= N) then i:=0; bBreak:=true; end_if;
    end_if;
    
  end_while;
  bBreak:=false;
  
  (* TEST *)
  if (Ix_local=0) then msg := LogMsg(MakeMsg(msg, 'END')); end_if; 

  (* Каждый час - рестарт счётчика в защиту от переполнения *)
  if (DTIME.ET > T#1h) then 
    PDT := CDT;
    DTIME(IN:=false);
    DTIME(IN:=true);
  end_if;
  return;

  {{__error:}}
  if (iErr = E_SUCCESS) then iErr := E_PROCESS; end_if;
  bRes := FALSE;
  bReStart := TRUE; (* Посылаем на рестарт *)
  
  (* Протоколирование ошибки *)
  msg:=LogMsg( MakeMsg('== PROCESS ERROR -> will be re-started! [ERR=', 
      Err2Str(iErr), ']'), Warning, iErr);
ELSE
  bRes := FALSE;
  bReStart := TRUE;
END_IF; (* IN *)
          
END_FUNCTION_BLOCK

(* Моделирование *)
PROGRAM P_MOD1
  VAR_EXTERNAL
    STAT : TStat;  (* Состояние выполнения *)
    F_Res : BOOL;  (* Флаг готовности результата *)
  END_VAR
  VAR
    CDT : DT;
    bRes : BOOL;
    Process_X1 : Process_XYZ;
    Process_X2 : Process_XYZ;
    Process_X0 : Process_XYZ;
  END_VAR
  VAR  (* added by the conversion: wires and edge detectors of the diagram *)
    _Do_PreProc19_ENO : BOOL;
    _Do_PreProc19_OUT : BOOL;
    _Do_PostProc37_ENO : BOOL;
    _Do_PostProc37_OUT : BOOL;
  END_VAR

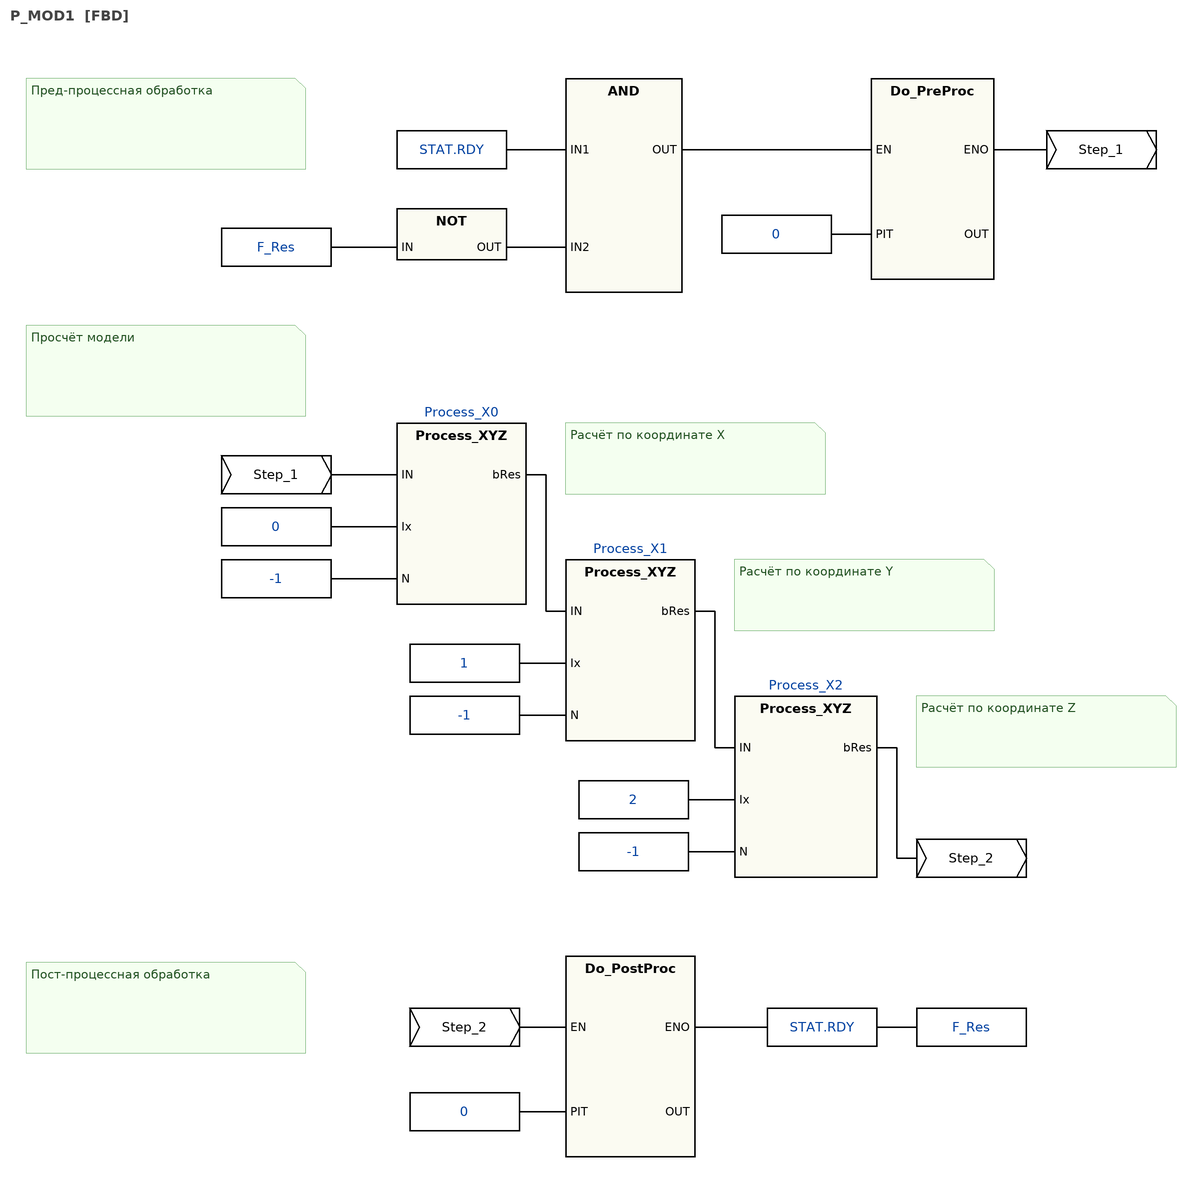
(* FBD diagram, written out as Structured Text *)
(* Пред-процессная обработка *)
(* Просчёт модели *)
(* Расчёт по координате X *)
(* Расчёт по координате Y *)
(* Расчёт по координате Z *)
(* Пост-процессная обработка *)
_Do_PreProc19_OUT := Do_PreProc(EN := STAT.RDY AND NOT F_Res, PIT := 0, ENO => _Do_PreProc19_ENO);
Process_X0(IN := _Do_PreProc19_ENO, Ix := 0, N := -1);
Process_X1(IN := Process_X0.bRes, Ix := 1, N := -1);
Process_X2(IN := Process_X1.bRes, Ix := 2, N := -1);
_Do_PostProc37_OUT := Do_PostProc(EN := Process_X2.bRes, PIT := 0, ENO => _Do_PostProc37_ENO);
STAT.RDY := _Do_PostProc37_ENO;
F_Res := STAT.RDY;
END_PROGRAM

(* Сборка буфера *)
PROGRAM P_MOD2
  VAR_EXTERNAL
    STS : TSets;
    MD460 : UDINT;
    MD461 : UDINT;
    MD462 : UDINT;
    MD463 : UDINT;
    MD464 : UDINT;
    MD465 : UDINT;
    MD466 : UDINT;
    MD467 : UDINT;
    MD468 : UDINT;
    MD469 : UDINT;
    MD470 : UDINT;
    MD471 : UDINT;
    MD472 : UDINT;
    MD473 : UDINT;
    MD474 : UDINT;
    MD475 : UDINT;
    MD476 : UDINT;
    MD477 : UDINT;
    MD478 : UDINT;
    MD479 : UDINT;
    MD480 : UDINT;
    MD481 : UDINT;
    MD482 : UDINT;
    MD483 : UDINT;
    MD484 : UDINT;
    MD485 : UDINT;
    MD486 : UDINT;
    MD487 : UDINT;
    MD488 : UDINT;
    MD489 : UDINT;
  END_VAR

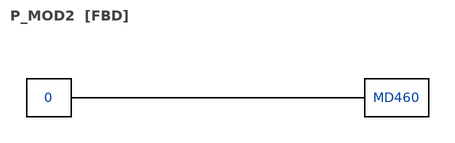
(* FBD diagram, written out as Structured Text *)
MD460 := 0;
END_PROGRAM

(* Заголовок из регистров *)
FUNCTION m_head : THead
  VAR_INPUT
    MD0 : UDINT;
    MD1 : UDINT;
    MD2 : UDINT;
    MD3 : UDINT;
    MD4 : UDINT;
    MD5 : UDINT;
    MD6 : UDINT;
    MD7 : UDINT;
    MD8 : UDINT;
    MD9 : UDINT;
  END_VAR

            m_head.Ni     := UINT_TO_SINT(UDINT_TO_UINT(MD0/65536)/256);            (* Количество элементов  *)
m_head.Ng     := UINT_TO_SINT(mod(UDINT_TO_UINT(MD0/65536),256));       (* Количество сеток      *)
m_head.Nm     := UINT_TO_SINT(UDINT_TO_UINT(mod(MD0,65536))/256);       (* Количество материалов *)
m_head.Nv     := UINT_TO_SINT(mod(UDINT_TO_UINT(mod(MD0,65536)),256));  (* Количество величин    *)
m_head.Np     := UINT_TO_SINT(UDINT_TO_UINT(MD1/65536)/256);            (* Количество профилей   *)
m_head.Ri     := UINT_TO_SINT(mod(UDINT_TO_UINT(MD1/65536),256));       (* Резерв                *)

m_head.ID     := UDINT_TO_UINT(mod(MD1,65536)); (* ID эл-та для выкладки сетки в регистры *)

m_head.TR[0]  := UDINT_TO_TIME(MD2); (* Период 1 *)
m_head.TR[1]  := UDINT_TO_TIME(MD3); (* Период 2 *)
m_head.TR[2]  := UDINT_TO_TIME(MD4); (* Период 3 *)
m_head.TR[3]  := UDINT_TO_TIME(MD5); (* Период 4 *)

m_head.Ax     := UDINT_TO_UINT(MD6/65536);      (* Направление перпендикуляра секущей *)
m_head.pX     := UDINT_TO_INT(mod(MD6,65536));  (* Координата X опорной точки секущей *)
m_head.pY     := UDINT_TO_INT(MD7/65536);       (* Координата Y опорной точки секущей *)
m_head.pZ     := UDINT_TO_INT(mod(MD7,65536));  (* Координата Z опорной точки секущей *)

m_head.RV[0]  := UDINT_TO_DINT(MD8); (* резерв *)
m_head.RV[1]  := UDINT_TO_DINT(MD9); (* резерв *)
          
END_FUNCTION

(* Чтение заголовка из регистров *)
FUNCTION_BLOCK GetHead
  VAR_EXTERNAL
    MD0 : UDINT;
    MD1 : UDINT;
    MD2 : UDINT;
    MD3 : UDINT;
    MD4 : UDINT;
    MD5 : UDINT;
    MD6 : UDINT;
    MD7 : UDINT;
    MD8 : UDINT;
    MD9 : UDINT;
  END_VAR
  VAR_OUTPUT
    HEAD : THead;
  END_VAR

            HEAD := m_head(MD0,MD1,MD2,MD3,MD4,MD5,MD6,MD7,MD8,MD9);

          
END_FUNCTION_BLOCK

(* Компоновка длинного целого *)
FUNCTION int4ul : ULINT
  VAR_INPUT
    I0 : INT;
    I1 : INT;
    I2 : INT;
    I3 : INT;
  END_VAR

            int4ul := INT_TO_ULINT(I0)*16#0001000000000000 + 
          INT_TO_ULINT(I1)*16#0000000100000000 +
          INT_TO_ULINT(I2)*16#0000000000010000 +
          INT_TO_ULINT(I3);
         

          
END_FUNCTION

(* Выкладка длинных целых (x4) *)
FUNCTION_BLOCK DistLong4
  VAR_INPUT
    LONG4 : ARRAY[0..3] OF ULINT;  (* Объект "массив 4x ULINT" *)
  END_VAR
  VAR_OUTPUT
    ML0 : ULINT;
    ML1 : ULINT;
    ML2 : ULINT;
    ML3 : ULINT;
  END_VAR

            ML0 := LONG4[0]; 
ML1 := LONG4[1]; 
ML2 := LONG4[2]; 
ML3 := LONG4[3]; 

          
END_FUNCTION_BLOCK

(* Запись элемента в выходные массивы *)
FUNCTION_BLOCK SetLong4
  VAR_EXTERNAL
    ML0 : ULINT;
    ML1 : ULINT;
    ML2 : ULINT;
    ML3 : ULINT;
    ML4 : ULINT;
    ML5 : ULINT;
    ML6 : ULINT;
    ML7 : ULINT;
    ML8 : ULINT;
    ML9 : ULINT;
    ML10 : ULINT;
    ML11 : ULINT;
    ML12 : ULINT;
    ML13 : ULINT;
    ML14 : ULINT;
    ML15 : ULINT;
    ML16 : ULINT;
    ML17 : ULINT;
    ML18 : ULINT;
    ML19 : ULINT;
    ML20 : ULINT;
    ML21 : ULINT;
    ML22 : ULINT;
    ML23 : ULINT;
    ML24 : ULINT;
    ML25 : ULINT;
    ML26 : ULINT;
    ML27 : ULINT;
    ML28 : ULINT;
    ML29 : ULINT;
    ML30 : ULINT;
    ML31 : ULINT;
    ML32 : ULINT;
    ML33 : ULINT;
    ML34 : ULINT;
    ML35 : ULINT;
    ML36 : ULINT;
    ML37 : ULINT;
    ML38 : ULINT;
    ML39 : ULINT;
    ML40 : ULINT;
    ML41 : ULINT;
    ML42 : ULINT;
    ML43 : ULINT;
    ML44 : ULINT;
    ML45 : ULINT;
    ML46 : ULINT;
    ML47 : ULINT;
    ML48 : ULINT;
    ML49 : ULINT;
    ML50 : ULINT;
    ML51 : ULINT;
    ML52 : ULINT;
    ML53 : ULINT;
    ML54 : ULINT;
    ML55 : ULINT;
    ML56 : ULINT;
    ML57 : ULINT;
    ML58 : ULINT;
    ML59 : ULINT;
    ML60 : ULINT;
    ML61 : ULINT;
    ML62 : ULINT;
    ML63 : ULINT;
    ML64 : ULINT;
    ML65 : ULINT;
    ML66 : ULINT;
    ML67 : ULINT;
    ML68 : ULINT;
    ML69 : ULINT;
    ML70 : ULINT;
    ML71 : ULINT;
    ML72 : ULINT;
    ML73 : ULINT;
    ML74 : ULINT;
    ML75 : ULINT;
    ML76 : ULINT;
    ML77 : ULINT;
    ML78 : ULINT;
    ML79 : ULINT;
    ML80 : ULINT;
    ML81 : ULINT;
    ML82 : ULINT;
    ML83 : ULINT;
    ML84 : ULINT;
    ML85 : ULINT;
    ML86 : ULINT;
    ML87 : ULINT;
    ML88 : ULINT;
    ML89 : ULINT;
    ML90 : ULINT;
    ML91 : ULINT;
    ML92 : ULINT;
    ML93 : ULINT;
    ML94 : ULINT;
    ML95 : ULINT;
    ML96 : ULINT;
    ML97 : ULINT;
    ML98 : ULINT;
    ML99 : ULINT;
    ML100 : ULINT;
    ML101 : ULINT;
    ML102 : ULINT;
    ML103 : ULINT;
    ML104 : ULINT;
    ML105 : ULINT;
    ML106 : ULINT;
    ML107 : ULINT;
    ML108 : ULINT;
    ML109 : ULINT;
    ML110 : ULINT;
    ML111 : ULINT;
    ML112 : ULINT;
    ML113 : ULINT;
    ML114 : ULINT;
    ML115 : ULINT;
    ML116 : ULINT;
    ML117 : ULINT;
    ML118 : ULINT;
    ML119 : ULINT;
    ML120 : ULINT;
    ML121 : ULINT;
    ML122 : ULINT;
    ML123 : ULINT;
    ML124 : ULINT;
    ML125 : ULINT;
    ML126 : ULINT;
    ML127 : ULINT;
    ML128 : ULINT;
    ML129 : ULINT;
    ML130 : ULINT;
    ML131 : ULINT;
    ML132 : ULINT;
    ML133 : ULINT;
    ML134 : ULINT;
    ML135 : ULINT;
    ML136 : ULINT;
    ML137 : ULINT;
    ML138 : ULINT;
    ML139 : ULINT;
    ML140 : ULINT;
    ML141 : ULINT;
    ML142 : ULINT;
    ML143 : ULINT;
    ML144 : ULINT;
    ML145 : ULINT;
    ML146 : ULINT;
    ML147 : ULINT;
    ML148 : ULINT;
    ML149 : ULINT;
    ML150 : ULINT;
    ML151 : ULINT;
    ML152 : ULINT;
    ML153 : ULINT;
    ML154 : ULINT;
    ML155 : ULINT;
    ML156 : ULINT;
    ML157 : ULINT;
    ML158 : ULINT;
    ML159 : ULINT;
    ML160 : ULINT;
    ML161 : ULINT;
    ML162 : ULINT;
    ML163 : ULINT;
    ML164 : ULINT;
    ML165 : ULINT;
    ML166 : ULINT;
    ML167 : ULINT;
    ML168 : ULINT;
    ML169 : ULINT;
    ML170 : ULINT;
    ML171 : ULINT;
    ML172 : ULINT;
    ML173 : ULINT;
    ML174 : ULINT;
    ML175 : ULINT;
    ML176 : ULINT;
    ML177 : ULINT;
    ML178 : ULINT;
    ML179 : ULINT;
    ML180 : ULINT;
    ML181 : ULINT;
    ML182 : ULINT;
    ML183 : ULINT;
    ML184 : ULINT;
    ML185 : ULINT;
    ML186 : ULINT;
    ML187 : ULINT;
    ML188 : ULINT;
    ML189 : ULINT;
    ML190 : ULINT;
    ML191 : ULINT;
    ML192 : ULINT;
    ML193 : ULINT;
    ML194 : ULINT;
    ML195 : ULINT;
    ML196 : ULINT;
    ML197 : ULINT;
    ML198 : ULINT;
    ML199 : ULINT;
    ML200 : ULINT;
    ML201 : ULINT;
    ML202 : ULINT;
    ML203 : ULINT;
    ML204 : ULINT;
    ML205 : ULINT;
    ML206 : ULINT;
    ML207 : ULINT;
    ML208 : ULINT;
    ML209 : ULINT;
    ML210 : ULINT;
    ML211 : ULINT;
    ML212 : ULINT;
    ML213 : ULINT;
    ML214 : ULINT;
    ML215 : ULINT;
    ML216 : ULINT;
    ML217 : ULINT;
    ML218 : ULINT;
    ML219 : ULINT;
    ML220 : ULINT;
    ML221 : ULINT;
    ML222 : ULINT;
    ML223 : ULINT;
    ML224 : ULINT;
    ML225 : ULINT;
    ML226 : ULINT;
    ML227 : ULINT;
    ML228 : ULINT;
    ML229 : ULINT;
    ML230 : ULINT;
    ML231 : ULINT;
    ML232 : ULINT;
    ML233 : ULINT;
    ML234 : ULINT;
    ML235 : ULINT;
    ML236 : ULINT;
    ML237 : ULINT;
    ML238 : ULINT;
    ML239 : ULINT;
    ML240 : ULINT;
    ML241 : ULINT;
    ML242 : ULINT;
    ML243 : ULINT;
    ML244 : ULINT;
    ML245 : ULINT;
    ML246 : ULINT;
    ML247 : ULINT;
    ML248 : ULINT;
    ML249 : ULINT;
    ML250 : ULINT;
    ML251 : ULINT;
    ML252 : ULINT;
    ML253 : ULINT;
    ML254 : ULINT;
    ML255 : ULINT;
    ML256 : ULINT;
    ML257 : ULINT;
    ML258 : ULINT;
    ML259 : ULINT;
    ML260 : ULINT;
    ML261 : ULINT;
    ML262 : ULINT;
    ML263 : ULINT;
    ML264 : ULINT;
    ML265 : ULINT;
    ML266 : ULINT;
    ML267 : ULINT;
    ML268 : ULINT;
    ML269 : ULINT;
    ML270 : ULINT;
    ML271 : ULINT;
    ML272 : ULINT;
    ML273 : ULINT;
    ML274 : ULINT;
    ML275 : ULINT;
    ML276 : ULINT;
    ML277 : ULINT;
    ML278 : ULINT;
    ML279 : ULINT;
    ML280 : ULINT;
    ML281 : ULINT;
    ML282 : ULINT;
    ML283 : ULINT;
    ML284 : ULINT;
    ML285 : ULINT;
    ML286 : ULINT;
    ML287 : ULINT;
    ML288 : ULINT;
    ML289 : ULINT;
    ML290 : ULINT;
    ML291 : ULINT;
    ML292 : ULINT;
    ML293 : ULINT;
    ML294 : ULINT;
    ML295 : ULINT;
    ML296 : ULINT;
    ML297 : ULINT;
    ML298 : ULINT;
    ML299 : ULINT;
    ML300 : ULINT;
    ML301 : ULINT;
    ML302 : ULINT;
    ML303 : ULINT;
    ML304 : ULINT;
    ML305 : ULINT;
    ML306 : ULINT;
    ML307 : ULINT;
    ML308 : ULINT;
    ML309 : ULINT;
    ML310 : ULINT;
    ML311 : ULINT;
    ML312 : ULINT;
    ML313 : ULINT;
    ML314 : ULINT;
    ML315 : ULINT;
    ML316 : ULINT;
    ML317 : ULINT;
    ML318 : ULINT;
    ML319 : ULINT;
    ML320 : ULINT;
    ML321 : ULINT;
    ML322 : ULINT;
    ML323 : ULINT;
    ML324 : ULINT;
    ML325 : ULINT;
    ML326 : ULINT;
    ML327 : ULINT;
    ML328 : ULINT;
    ML329 : ULINT;
    ML330 : ULINT;
    ML331 : ULINT;
    ML332 : ULINT;
    ML333 : ULINT;
    ML334 : ULINT;
    ML335 : ULINT;
    ML336 : ULINT;
    ML337 : ULINT;
    ML338 : ULINT;
    ML339 : ULINT;
    ML340 : ULINT;
    ML341 : ULINT;
    ML342 : ULINT;
    ML343 : ULINT;
    ML344 : ULINT;
    ML345 : ULINT;
    ML346 : ULINT;
    ML347 : ULINT;
    ML348 : ULINT;
    ML349 : ULINT;
    ML350 : ULINT;
    ML351 : ULINT;
    ML352 : ULINT;
    ML353 : ULINT;
    ML354 : ULINT;
    ML355 : ULINT;
    ML356 : ULINT;
    ML357 : ULINT;
    ML358 : ULINT;
    ML359 : ULINT;
    ML360 : ULINT;
    ML361 : ULINT;
    ML362 : ULINT;
    ML363 : ULINT;
    ML364 : ULINT;
    ML365 : ULINT;
    ML366 : ULINT;
    ML367 : ULINT;
    ML368 : ULINT;
    ML369 : ULINT;
    ML370 : ULINT;
    ML371 : ULINT;
    ML372 : ULINT;
    ML373 : ULINT;
    ML374 : ULINT;
    ML375 : ULINT;
    ML376 : ULINT;
    ML377 : ULINT;
    ML378 : ULINT;
    ML379 : ULINT;
    ML380 : ULINT;
    ML381 : ULINT;
    ML382 : ULINT;
    ML383 : ULINT;
    ML384 : ULINT;
    ML385 : ULINT;
    ML386 : ULINT;
    ML387 : ULINT;
    ML388 : ULINT;
    ML389 : ULINT;
    ML390 : ULINT;
    ML391 : ULINT;
    ML392 : ULINT;
    ML393 : ULINT;
    ML394 : ULINT;
    ML395 : ULINT;
    ML396 : ULINT;
    ML397 : ULINT;
    ML398 : ULINT;
    ML399 : ULINT;
    ML400 : ULINT;
    ML401 : ULINT;
    ML402 : ULINT;
    ML403 : ULINT;
    ML404 : ULINT;
    ML405 : ULINT;
    ML406 : ULINT;
    ML407 : ULINT;
    ML408 : ULINT;
    ML409 : ULINT;
    ML410 : ULINT;
    ML411 : ULINT;
    ML412 : ULINT;
    ML413 : ULINT;
    ML414 : ULINT;
    ML415 : ULINT;
    ML416 : ULINT;
    ML417 : ULINT;
    ML418 : ULINT;
    ML419 : ULINT;
    ML420 : ULINT;
    ML421 : ULINT;
    ML422 : ULINT;
    ML423 : ULINT;
    ML424 : ULINT;
    ML425 : ULINT;
    ML426 : ULINT;
    ML427 : ULINT;
    ML428 : ULINT;
    ML429 : ULINT;
    ML430 : ULINT;
    ML431 : ULINT;
    ML432 : ULINT;
    ML433 : ULINT;
    ML434 : ULINT;
    ML435 : ULINT;
    ML436 : ULINT;
    ML437 : ULINT;
    ML438 : ULINT;
    ML439 : ULINT;
    ML440 : ULINT;
    ML441 : ULINT;
    ML442 : ULINT;
    ML443 : ULINT;
    ML444 : ULINT;
    ML445 : ULINT;
    ML446 : ULINT;
    ML447 : ULINT;
    ML448 : ULINT;
    ML449 : ULINT;
    ML450 : ULINT;
    ML451 : ULINT;
    ML452 : ULINT;
    ML453 : ULINT;
    ML454 : ULINT;
    ML455 : ULINT;
    ML456 : ULINT;
    ML457 : ULINT;
    ML458 : ULINT;
    ML459 : ULINT;
    ML460 : ULINT;
    ML461 : ULINT;
    ML462 : ULINT;
    ML463 : ULINT;
    ML464 : ULINT;
    ML465 : ULINT;
    ML466 : ULINT;
    ML467 : ULINT;
    ML468 : ULINT;
    ML469 : ULINT;
    ML470 : ULINT;
    ML471 : ULINT;
    ML472 : ULINT;
    ML473 : ULINT;
    ML474 : ULINT;
    ML475 : ULINT;
    ML476 : ULINT;
    ML477 : ULINT;
    ML478 : ULINT;
    ML479 : ULINT;
    ML480 : ULINT;
    ML481 : ULINT;
    ML482 : ULINT;
    ML483 : ULINT;
    ML484 : ULINT;
    ML485 : ULINT;
    ML486 : ULINT;
    ML487 : ULINT;
    ML488 : ULINT;
    ML489 : ULINT;
    ML490 : ULINT;
    ML491 : ULINT;
    ML492 : ULINT;
    ML493 : ULINT;
    ML494 : ULINT;
    ML495 : ULINT;
    ML496 : ULINT;
    ML497 : ULINT;
    ML498 : ULINT;
    ML499 : ULINT;
    ML500 : ULINT;
    ML501 : ULINT;
    ML502 : ULINT;
    ML503 : ULINT;
    ML504 : ULINT;
    ML505 : ULINT;
    ML506 : ULINT;
    ML507 : ULINT;
    ML508 : ULINT;
    ML509 : ULINT;
    ML510 : ULINT;
    ML511 : ULINT;
    ML512 : ULINT;
    ML513 : ULINT;
    ML514 : ULINT;
    ML515 : ULINT;
    ML516 : ULINT;
    ML517 : ULINT;
    ML518 : ULINT;
    ML519 : ULINT;
    ML520 : ULINT;
    ML521 : ULINT;
    ML522 : ULINT;
    ML523 : ULINT;
    ML524 : ULINT;
    ML525 : ULINT;
    ML526 : ULINT;
    ML527 : ULINT;
    ML528 : ULINT;
    ML529 : ULINT;
    ML530 : ULINT;
    ML531 : ULINT;
    ML532 : ULINT;
    ML533 : ULINT;
    ML534 : ULINT;
    ML535 : ULINT;
    ML536 : ULINT;
    ML537 : ULINT;
    ML538 : ULINT;
    ML539 : ULINT;
    ML540 : ULINT;
    ML541 : ULINT;
    ML542 : ULINT;
    ML543 : ULINT;
    ML544 : ULINT;
    ML545 : ULINT;
    ML546 : ULINT;
    ML547 : ULINT;
    ML548 : ULINT;
    ML549 : ULINT;
    ML550 : ULINT;
    ML551 : ULINT;
    ML552 : ULINT;
    ML553 : ULINT;
    ML554 : ULINT;
    ML555 : ULINT;
    ML556 : ULINT;
    ML557 : ULINT;
    ML558 : ULINT;
    ML559 : ULINT;
    ML560 : ULINT;
    ML561 : ULINT;
    ML562 : ULINT;
    ML563 : ULINT;
    ML564 : ULINT;
    ML565 : ULINT;
    ML566 : ULINT;
    ML567 : ULINT;
    ML568 : ULINT;
    ML569 : ULINT;
    ML570 : ULINT;
    ML571 : ULINT;
    ML572 : ULINT;
    ML573 : ULINT;
    ML574 : ULINT;
    ML575 : ULINT;
    ML576 : ULINT;
    ML577 : ULINT;
    ML578 : ULINT;
    ML579 : ULINT;
    ML580 : ULINT;
    ML581 : ULINT;
    ML582 : ULINT;
    ML583 : ULINT;
    ML584 : ULINT;
    ML585 : ULINT;
    ML586 : ULINT;
    ML587 : ULINT;
    ML588 : ULINT;
    ML589 : ULINT;
    ML590 : ULINT;
    ML591 : ULINT;
    ML592 : ULINT;
    ML593 : ULINT;
    ML594 : ULINT;
    ML595 : ULINT;
    ML596 : ULINT;
    ML597 : ULINT;
    ML598 : ULINT;
    ML599 : ULINT;
    ML600 : ULINT;
    ML601 : ULINT;
    ML602 : ULINT;
    ML603 : ULINT;
    ML604 : ULINT;
    ML605 : ULINT;
    ML606 : ULINT;
    ML607 : ULINT;
    ML608 : ULINT;
    ML609 : ULINT;
    ML610 : ULINT;
    ML611 : ULINT;
    ML612 : ULINT;
    ML613 : ULINT;
    ML614 : ULINT;
    ML615 : ULINT;
    ML616 : ULINT;
    ML617 : ULINT;
    ML618 : ULINT;
    ML619 : ULINT;
    ML620 : ULINT;
    ML621 : ULINT;
    ML622 : ULINT;
    ML623 : ULINT;
    ML624 : ULINT;
    ML625 : ULINT;
    ML626 : ULINT;
    ML627 : ULINT;
    ML628 : ULINT;
    ML629 : ULINT;
    ML630 : ULINT;
    ML631 : ULINT;
    ML632 : ULINT;
    ML633 : ULINT;
    ML634 : ULINT;
    ML635 : ULINT;
    ML636 : ULINT;
    ML637 : ULINT;
    ML638 : ULINT;
    ML639 : ULINT;
    ML640 : ULINT;
    ML641 : ULINT;
    ML642 : ULINT;
    ML643 : ULINT;
    ML644 : ULINT;
    ML645 : ULINT;
    ML646 : ULINT;
    ML647 : ULINT;
    ML648 : ULINT;
    ML649 : ULINT;
    ML650 : ULINT;
    ML651 : ULINT;
    ML652 : ULINT;
    ML653 : ULINT;
    ML654 : ULINT;
    ML655 : ULINT;
    ML656 : ULINT;
    ML657 : ULINT;
    ML658 : ULINT;
    ML659 : ULINT;
    ML660 : ULINT;
    ML661 : ULINT;
    ML662 : ULINT;
    ML663 : ULINT;
    ML664 : ULINT;
    ML665 : ULINT;
    ML666 : ULINT;
    ML667 : ULINT;
    ML668 : ULINT;
    ML669 : ULINT;
    ML670 : ULINT;
    ML671 : ULINT;
    ML672 : ULINT;
    ML673 : ULINT;
    ML674 : ULINT;
    ML675 : ULINT;
    ML676 : ULINT;
    ML677 : ULINT;
    ML678 : ULINT;
    ML679 : ULINT;
    ML680 : ULINT;
    ML681 : ULINT;
    ML682 : ULINT;
    ML683 : ULINT;
    ML684 : ULINT;
    ML685 : ULINT;
    ML686 : ULINT;
    ML687 : ULINT;
    ML688 : ULINT;
    ML689 : ULINT;
    ML690 : ULINT;
    ML691 : ULINT;
    ML692 : ULINT;
    ML693 : ULINT;
    ML694 : ULINT;
    ML695 : ULINT;
    ML696 : ULINT;
    ML697 : ULINT;
    ML698 : ULINT;
    ML699 : ULINT;
    ML700 : ULINT;
    ML701 : ULINT;
    ML702 : ULINT;
    ML703 : ULINT;
    ML704 : ULINT;
    ML705 : ULINT;
    ML706 : ULINT;
    ML707 : ULINT;
    ML708 : ULINT;
    ML709 : ULINT;
    ML710 : ULINT;
    ML711 : ULINT;
    ML712 : ULINT;
    ML713 : ULINT;
    ML714 : ULINT;
    ML715 : ULINT;
    ML716 : ULINT;
    ML717 : ULINT;
    ML718 : ULINT;
    ML719 : ULINT;
    ML720 : ULINT;
    ML721 : ULINT;
    ML722 : ULINT;
    ML723 : ULINT;
    ML724 : ULINT;
    ML725 : ULINT;
    ML726 : ULINT;
    ML727 : ULINT;
    ML728 : ULINT;
    ML729 : ULINT;
    ML730 : ULINT;
    ML731 : ULINT;
    ML732 : ULINT;
    ML733 : ULINT;
    ML734 : ULINT;
    ML735 : ULINT;
    ML736 : ULINT;
    ML737 : ULINT;
    ML738 : ULINT;
    ML739 : ULINT;
    ML740 : ULINT;
    ML741 : ULINT;
    ML742 : ULINT;
    ML743 : ULINT;
    ML744 : ULINT;
    ML745 : ULINT;
    ML746 : ULINT;
    ML747 : ULINT;
    ML748 : ULINT;
    ML749 : ULINT;
    ML750 : ULINT;
    ML751 : ULINT;
    ML752 : ULINT;
    ML753 : ULINT;
    ML754 : ULINT;
    ML755 : ULINT;
    ML756 : ULINT;
    ML757 : ULINT;
    ML758 : ULINT;
    ML759 : ULINT;
    ML760 : ULINT;
    ML761 : ULINT;
    ML762 : ULINT;
    ML763 : ULINT;
    ML764 : ULINT;
    ML765 : ULINT;
    ML766 : ULINT;
    ML767 : ULINT;
    ML768 : ULINT;
    ML769 : ULINT;
    ML770 : ULINT;
    ML771 : ULINT;
    ML772 : ULINT;
    ML773 : ULINT;
    ML774 : ULINT;
    ML775 : ULINT;
    ML776 : ULINT;
    ML777 : ULINT;
    ML778 : ULINT;
    ML779 : ULINT;
    ML780 : ULINT;
    ML781 : ULINT;
    ML782 : ULINT;
    ML783 : ULINT;
    ML784 : ULINT;
    ML785 : ULINT;
    ML786 : ULINT;
    ML787 : ULINT;
    ML788 : ULINT;
    ML789 : ULINT;
    ML790 : ULINT;
    ML791 : ULINT;
    ML792 : ULINT;
    ML793 : ULINT;
    ML794 : ULINT;
    ML795 : ULINT;
    ML796 : ULINT;
    ML797 : ULINT;
    ML798 : ULINT;
    ML799 : ULINT;
    ML800 : ULINT;
    ML801 : ULINT;
    ML802 : ULINT;
    ML803 : ULINT;
    ML804 : ULINT;
    ML805 : ULINT;
    ML806 : ULINT;
    ML807 : ULINT;
    ML808 : ULINT;
    ML809 : ULINT;
    ML810 : ULINT;
    ML811 : ULINT;
    ML812 : ULINT;
    ML813 : ULINT;
    ML814 : ULINT;
    ML815 : ULINT;
    ML816 : ULINT;
    ML817 : ULINT;
    ML818 : ULINT;
    ML819 : ULINT;
    ML820 : ULINT;
    ML821 : ULINT;
    ML822 : ULINT;
    ML823 : ULINT;
    ML824 : ULINT;
    ML825 : ULINT;
    ML826 : ULINT;
    ML827 : ULINT;
    ML828 : ULINT;
    ML829 : ULINT;
    ML830 : ULINT;
    ML831 : ULINT;
    ML832 : ULINT;
    ML833 : ULINT;
    ML834 : ULINT;
    ML835 : ULINT;
    ML836 : ULINT;
    ML837 : ULINT;
    ML838 : ULINT;
    ML839 : ULINT;
    ML840 : ULINT;
    ML841 : ULINT;
    ML842 : ULINT;
    ML843 : ULINT;
    ML844 : ULINT;
    ML845 : ULINT;
    ML846 : ULINT;
    ML847 : ULINT;
    ML848 : ULINT;
    ML849 : ULINT;
    ML850 : ULINT;
    ML851 : ULINT;
    ML852 : ULINT;
    ML853 : ULINT;
    ML854 : ULINT;
    ML855 : ULINT;
    ML856 : ULINT;
    ML857 : ULINT;
    ML858 : ULINT;
    ML859 : ULINT;
    ML860 : ULINT;
    ML861 : ULINT;
    ML862 : ULINT;
    ML863 : ULINT;
    ML864 : ULINT;
    ML865 : ULINT;
    ML866 : ULINT;
    ML867 : ULINT;
    ML868 : ULINT;
    ML869 : ULINT;
    ML870 : ULINT;
    ML871 : ULINT;
    ML872 : ULINT;
    ML873 : ULINT;
    ML874 : ULINT;
    ML875 : ULINT;
    ML876 : ULINT;
    ML877 : ULINT;
    ML878 : ULINT;
    ML879 : ULINT;
    ML880 : ULINT;
    ML881 : ULINT;
    ML882 : ULINT;
    ML883 : ULINT;
    ML884 : ULINT;
    ML885 : ULINT;
    ML886 : ULINT;
    ML887 : ULINT;
    ML888 : ULINT;
    ML889 : ULINT;
    ML890 : ULINT;
    ML891 : ULINT;
    ML892 : ULINT;
    ML893 : ULINT;
    ML894 : ULINT;
    ML895 : ULINT;
    ML896 : ULINT;
    ML897 : ULINT;
    ML898 : ULINT;
    ML899 : ULINT;
    ML900 : ULINT;
    ML901 : ULINT;
    ML902 : ULINT;
    ML903 : ULINT;
    ML904 : ULINT;
    ML905 : ULINT;
    ML906 : ULINT;
    ML907 : ULINT;
    ML908 : ULINT;
    ML909 : ULINT;
    ML910 : ULINT;
    ML911 : ULINT;
    ML912 : ULINT;
    ML913 : ULINT;
    ML914 : ULINT;
    ML915 : ULINT;
    ML916 : ULINT;
    ML917 : ULINT;
    ML918 : ULINT;
    ML919 : ULINT;
    ML920 : ULINT;
    ML921 : ULINT;
    ML922 : ULINT;
    ML923 : ULINT;
    ML924 : ULINT;
    ML925 : ULINT;
    ML926 : ULINT;
    ML927 : ULINT;
    ML928 : ULINT;
    ML929 : ULINT;
    ML930 : ULINT;
    ML931 : ULINT;
    ML932 : ULINT;
    ML933 : ULINT;
    ML934 : ULINT;
    ML935 : ULINT;
    ML936 : ULINT;
    ML937 : ULINT;
    ML938 : ULINT;
    ML939 : ULINT;
    ML940 : ULINT;
    ML941 : ULINT;
    ML942 : ULINT;
    ML943 : ULINT;
    ML944 : ULINT;
    ML945 : ULINT;
    ML946 : ULINT;
    ML947 : ULINT;
    ML948 : ULINT;
    ML949 : ULINT;
    ML950 : ULINT;
    ML951 : ULINT;
    ML952 : ULINT;
    ML953 : ULINT;
    ML954 : ULINT;
    ML955 : ULINT;
    ML956 : ULINT;
    ML957 : ULINT;
    ML958 : ULINT;
    ML959 : ULINT;
    ML960 : ULINT;
    ML961 : ULINT;
    ML962 : ULINT;
    ML963 : ULINT;
    ML964 : ULINT;
    ML965 : ULINT;
    ML966 : ULINT;
    ML967 : ULINT;
    ML968 : ULINT;
    ML969 : ULINT;
    ML970 : ULINT;
    ML971 : ULINT;
    ML972 : ULINT;
    ML973 : ULINT;
    ML974 : ULINT;
    ML975 : ULINT;
    ML976 : ULINT;
    ML977 : ULINT;
    ML978 : ULINT;
    ML979 : ULINT;
    ML980 : ULINT;
    ML981 : ULINT;
    ML982 : ULINT;
    ML983 : ULINT;
    ML984 : ULINT;
    ML985 : ULINT;
    ML986 : ULINT;
    ML987 : ULINT;
    ML988 : ULINT;
    ML989 : ULINT;
    ML990 : ULINT;
    ML991 : ULINT;
    ML992 : ULINT;
    ML993 : ULINT;
    ML994 : ULINT;
    ML995 : ULINT;
    ML996 : ULINT;
    ML997 : ULINT;
    ML998 : ULINT;
    ML999 : ULINT;
    ML1000 : ULINT;
    ML1001 : ULINT;
    ML1002 : ULINT;
    ML1003 : ULINT;
    ML1004 : ULINT;
    ML1005 : ULINT;
    ML1006 : ULINT;
    ML1007 : ULINT;
    ML1008 : ULINT;
    ML1009 : ULINT;
    ML1010 : ULINT;
    ML1011 : ULINT;
    ML1012 : ULINT;
    ML1013 : ULINT;
    ML1014 : ULINT;
    ML1015 : ULINT;
    ML1016 : ULINT;
    ML1017 : ULINT;
    ML1018 : ULINT;
    ML1019 : ULINT;
    ML1020 : ULINT;
    ML1021 : ULINT;
    ML1022 : ULINT;
    ML1023 : ULINT;
  END_VAR
  VAR_INPUT
    I : INT := 0;  (* Индекс в массиве ML [0..1023] *)
    LONG4 : ARRAY[0..3] OF ULINT;  (* Записываемое значение *)
  END_VAR
  VAR
    DIST : DistLong4;
  END_VAR

            CASE I OF
0:  DIST(LONG4:=LONG4, ML0=>ML0,  ML1=>ML1,  ML2=>ML2,  ML3=>ML3);
1:  DIST(LONG4:=LONG4, ML0=>ML4,  ML1=>ML5,  ML2=>ML6,  ML3=>ML7);
2:  DIST(LONG4:=LONG4, ML0=>ML8,  ML1=>ML9,  ML2=>ML10, ML3=>ML11);
3:  DIST(LONG4:=LONG4, ML0=>ML12, ML1=>ML13, ML2=>ML14, ML3=>ML15);
4:  DIST(LONG4:=LONG4, ML0=>ML16, ML1=>ML17, ML2=>ML18, ML3=>ML19);
5:  DIST(LONG4:=LONG4, ML0=>ML20, ML1=>ML21, ML2=>ML22, ML3=>ML23);
6:  DIST(LONG4:=LONG4, ML0=>ML24, ML1=>ML25, ML2=>ML26, ML3=>ML27);
7:  DIST(LONG4:=LONG4, ML0=>ML28, ML1=>ML29, ML2=>ML30, ML3=>ML31);
8:  DIST(LONG4:=LONG4, ML0=>ML32, ML1=>ML33, ML2=>ML34, ML3=>ML35);
9:  DIST(LONG4:=LONG4, ML0=>ML36, ML1=>ML37, ML2=>ML38, ML3=>ML39);
10: DIST(LONG4:=LONG4, ML0=>ML40, ML1=>ML41, ML2=>ML42, ML3=>ML43);
11: DIST(LONG4:=LONG4, ML0=>ML44, ML1=>ML45, ML2=>ML46, ML3=>ML47);
12: DIST(LONG4:=LONG4, ML0=>ML48, ML1=>ML49, ML2=>ML50, ML3=>ML51);
13: DIST(LONG4:=LONG4, ML0=>ML52, ML1=>ML53, ML2=>ML54, ML3=>ML55);
14: DIST(LONG4:=LONG4, ML0=>ML56, ML1=>ML57, ML2=>ML58, ML3=>ML59);
15: DIST(LONG4:=LONG4, ML0=>ML60, ML1=>ML61, ML2=>ML62, ML3=>ML63);
16: DIST(LONG4:=LONG4, ML0=>ML64, ML1=>ML65, ML2=>ML66, ML3=>ML67);
17: DIST(LONG4:=LONG4, ML0=>ML68, ML1=>ML69, ML2=>ML70, ML3=>ML71);
18: DIST(LONG4:=LONG4, ML0=>ML72, ML1=>ML73, ML2=>ML74, ML3=>ML75);
19: DIST(LONG4:=LONG4, ML0=>ML76, ML1=>ML77, ML2=>ML78, ML3=>ML79);
20: DIST(LONG4:=LONG4, ML0=>ML80, ML1=>ML81, ML2=>ML82, ML3=>ML83);
21: DIST(LONG4:=LONG4, ML0=>ML84, ML1=>ML85, ML2=>ML86, ML3=>ML87);
22: DIST(LONG4:=LONG4, ML0=>ML88, ML1=>ML89, ML2=>ML90, ML3=>ML91);
23: DIST(LONG4:=LONG4, ML0=>ML92, ML1=>ML93, ML2=>ML94, ML3=>ML95);
24: DIST(LONG4:=LONG4, ML0=>ML96, ML1=>ML97, ML2=>ML98, ML3=>ML99);
25: DIST(LONG4:=LONG4, ML0=>ML100, ML1=>ML101, ML2=>ML102, ML3=>ML103);
26: DIST(LONG4:=LONG4, ML0=>ML104, ML1=>ML105, ML2=>ML106, ML3=>ML107);
27: DIST(LONG4:=LONG4, ML0=>ML108, ML1=>ML109, ML2=>ML110, ML3=>ML111);
28: DIST(LONG4:=LONG4, ML0=>ML112, ML1=>ML113, ML2=>ML114, ML3=>ML115);
29: DIST(LONG4:=LONG4, ML0=>ML116, ML1=>ML117, ML2=>ML118, ML3=>ML119);
30: DIST(LONG4:=LONG4, ML0=>ML120, ML1=>ML121, ML2=>ML122, ML3=>ML123);
31: DIST(LONG4:=LONG4, ML0=>ML124, ML1=>ML125, ML2=>ML126, ML3=>ML127);
32: DIST(LONG4:=LONG4, ML0=>ML128, ML1=>ML129, ML2=>ML130, ML3=>ML131);
33: DIST(LONG4:=LONG4, ML0=>ML132, ML1=>ML133, ML2=>ML134, ML3=>ML135);
34: DIST(LONG4:=LONG4, ML0=>ML136, ML1=>ML137, ML2=>ML138, ML3=>ML139);
35: DIST(LONG4:=LONG4, ML0=>ML140, ML1=>ML141, ML2=>ML142, ML3=>ML143);
36: DIST(LONG4:=LONG4, ML0=>ML144, ML1=>ML145, ML2=>ML146, ML3=>ML147);
37: DIST(LONG4:=LONG4, ML0=>ML148, ML1=>ML149, ML2=>ML150, ML3=>ML151);
38: DIST(LONG4:=LONG4, ML0=>ML152, ML1=>ML153, ML2=>ML154, ML3=>ML155);
39: DIST(LONG4:=LONG4, ML0=>ML156, ML1=>ML157, ML2=>ML158, ML3=>ML159);
40: DIST(LONG4:=LONG4, ML0=>ML160, ML1=>ML161, ML2=>ML162, ML3=>ML163);
41: DIST(LONG4:=LONG4, ML0=>ML164, ML1=>ML165, ML2=>ML166, ML3=>ML167);
42: DIST(LONG4:=LONG4, ML0=>ML168, ML1=>ML169, ML2=>ML170, ML3=>ML171);
43: DIST(LONG4:=LONG4, ML0=>ML172, ML1=>ML173, ML2=>ML174, ML3=>ML175);
44: DIST(LONG4:=LONG4, ML0=>ML176, ML1=>ML177, ML2=>ML178, ML3=>ML179);
45: DIST(LONG4:=LONG4, ML0=>ML180, ML1=>ML181, ML2=>ML182, ML3=>ML183);
46: DIST(LONG4:=LONG4, ML0=>ML184, ML1=>ML185, ML2=>ML186, ML3=>ML187);
47: DIST(LONG4:=LONG4, ML0=>ML188, ML1=>ML189, ML2=>ML190, ML3=>ML191);
48: DIST(LONG4:=LONG4, ML0=>ML192, ML1=>ML193, ML2=>ML194, ML3=>ML195);
49: DIST(LONG4:=LONG4, ML0=>ML196, ML1=>ML197, ML2=>ML198, ML3=>ML199);
50: DIST(LONG4:=LONG4, ML0=>ML200, ML1=>ML201, ML2=>ML202, ML3=>ML203);
51: DIST(LONG4:=LONG4, ML0=>ML204, ML1=>ML205, ML2=>ML206, ML3=>ML207);
52: DIST(LONG4:=LONG4, ML0=>ML208, ML1=>ML209, ML2=>ML210, ML3=>ML211);
53: DIST(LONG4:=LONG4, ML0=>ML212, ML1=>ML213, ML2=>ML214, ML3=>ML215);
54: DIST(LONG4:=LONG4, ML0=>ML216, ML1=>ML217, ML2=>ML218, ML3=>ML219);
55: DIST(LONG4:=LONG4, ML0=>ML220, ML1=>ML221, ML2=>ML222, ML3=>ML223);
56: DIST(LONG4:=LONG4, ML0=>ML224, ML1=>ML225, ML2=>ML226, ML3=>ML227);
57: DIST(LONG4:=LONG4, ML0=>ML228, ML1=>ML229, ML2=>ML230, ML3=>ML231);
58: DIST(LONG4:=LONG4, ML0=>ML232, ML1=>ML233, ML2=>ML234, ML3=>ML235);
59: DIST(LONG4:=LONG4, ML0=>ML236, ML1=>ML237, ML2=>ML238, ML3=>ML239);
60: DIST(LONG4:=LONG4, ML0=>ML240, ML1=>ML241, ML2=>ML242, ML3=>ML243);
61: DIST(LONG4:=LONG4, ML0=>ML244, ML1=>ML245, ML2=>ML246, ML3=>ML247);
62: DIST(LONG4:=LONG4, ML0=>ML248, ML1=>ML249, ML2=>ML250, ML3=>ML251);
63: DIST(LONG4:=LONG4, ML0=>ML252, ML1=>ML253, ML2=>ML254, ML3=>ML255);
64: DIST(LONG4:=LONG4, ML0=>ML256, ML1=>ML257, ML2=>ML258, ML3=>ML259);
65: DIST(LONG4:=LONG4, ML0=>ML260, ML1=>ML261, ML2=>ML262, ML3=>ML263);
66: DIST(LONG4:=LONG4, ML0=>ML264, ML1=>ML265, ML2=>ML266, ML3=>ML267);
67: DIST(LONG4:=LONG4, ML0=>ML268, ML1=>ML269, ML2=>ML270, ML3=>ML271);
68: DIST(LONG4:=LONG4, ML0=>ML272, ML1=>ML273, ML2=>ML274, ML3=>ML275);
69: DIST(LONG4:=LONG4, ML0=>ML276, ML1=>ML277, ML2=>ML278, ML3=>ML279);
70: DIST(LONG4:=LONG4, ML0=>ML280, ML1=>ML281, ML2=>ML282, ML3=>ML283);
71: DIST(LONG4:=LONG4, ML0=>ML284, ML1=>ML285, ML2=>ML286, ML3=>ML287);
72: DIST(LONG4:=LONG4, ML0=>ML288, ML1=>ML289, ML2=>ML290, ML3=>ML291);
73: DIST(LONG4:=LONG4, ML0=>ML292, ML1=>ML293, ML2=>ML294, ML3=>ML295);
74: DIST(LONG4:=LONG4, ML0=>ML296, ML1=>ML297, ML2=>ML298, ML3=>ML299);
75: DIST(LONG4:=LONG4, ML0=>ML300, ML1=>ML301, ML2=>ML302, ML3=>ML303);
76: DIST(LONG4:=LONG4, ML0=>ML304, ML1=>ML305, ML2=>ML306, ML3=>ML307);
77: DIST(LONG4:=LONG4, ML0=>ML308, ML1=>ML309, ML2=>ML310, ML3=>ML311);
78: DIST(LONG4:=LONG4, ML0=>ML312, ML1=>ML313, ML2=>ML314, ML3=>ML315);
79: DIST(LONG4:=LONG4, ML0=>ML316, ML1=>ML317, ML2=>ML318, ML3=>ML319);
80: DIST(LONG4:=LONG4, ML0=>ML320, ML1=>ML321, ML2=>ML322, ML3=>ML323);
81: DIST(LONG4:=LONG4, ML0=>ML324, ML1=>ML325, ML2=>ML326, ML3=>ML327);
82: DIST(LONG4:=LONG4, ML0=>ML328, ML1=>ML329, ML2=>ML330, ML3=>ML331);
83: DIST(LONG4:=LONG4, ML0=>ML332, ML1=>ML333, ML2=>ML334, ML3=>ML335);
84: DIST(LONG4:=LONG4, ML0=>ML336, ML1=>ML337, ML2=>ML338, ML3=>ML339);
85: DIST(LONG4:=LONG4, ML0=>ML340, ML1=>ML341, ML2=>ML342, ML3=>ML343);
86: DIST(LONG4:=LONG4, ML0=>ML344, ML1=>ML345, ML2=>ML346, ML3=>ML347);
87: DIST(LONG4:=LONG4, ML0=>ML348, ML1=>ML349, ML2=>ML350, ML3=>ML351);
88: DIST(LONG4:=LONG4, ML0=>ML352, ML1=>ML353, ML2=>ML354, ML3=>ML355);
89: DIST(LONG4:=LONG4, ML0=>ML356, ML1=>ML357, ML2=>ML358, ML3=>ML359);
90: DIST(LONG4:=LONG4, ML0=>ML360, ML1=>ML361, ML2=>ML362, ML3=>ML363);
91: DIST(LONG4:=LONG4, ML0=>ML364, ML1=>ML365, ML2=>ML366, ML3=>ML367);
92: DIST(LONG4:=LONG4, ML0=>ML368, ML1=>ML369, ML2=>ML370, ML3=>ML371);
93: DIST(LONG4:=LONG4, ML0=>ML372, ML1=>ML373, ML2=>ML374, ML3=>ML375);
94: DIST(LONG4:=LONG4, ML0=>ML376, ML1=>ML377, ML2=>ML378, ML3=>ML379);
95: DIST(LONG4:=LONG4, ML0=>ML380, ML1=>ML381, ML2=>ML382, ML3=>ML383);
96: DIST(LONG4:=LONG4, ML0=>ML384, ML1=>ML385, ML2=>ML386, ML3=>ML387);
97: DIST(LONG4:=LONG4, ML0=>ML388, ML1=>ML389, ML2=>ML390, ML3=>ML391);
98: DIST(LONG4:=LONG4, ML0=>ML392, ML1=>ML393, ML2=>ML394, ML3=>ML395);
99: DIST(LONG4:=LONG4, ML0=>ML396, ML1=>ML397, ML2=>ML398, ML3=>ML399);
100: DIST(LONG4:=LONG4, ML0=>ML400, ML1=>ML401, ML2=>ML402, ML3=>ML403);
101: DIST(LONG4:=LONG4, ML0=>ML404, ML1=>ML405, ML2=>ML406, ML3=>ML407);
102: DIST(LONG4:=LONG4, ML0=>ML408, ML1=>ML409, ML2=>ML410, ML3=>ML411);
103: DIST(LONG4:=LONG4, ML0=>ML412, ML1=>ML413, ML2=>ML414, ML3=>ML415);
104: DIST(LONG4:=LONG4, ML0=>ML416, ML1=>ML417, ML2=>ML418, ML3=>ML419);
105: DIST(LONG4:=LONG4, ML0=>ML420, ML1=>ML421, ML2=>ML422, ML3=>ML423);
106: DIST(LONG4:=LONG4, ML0=>ML424, ML1=>ML425, ML2=>ML426, ML3=>ML427);
107: DIST(LONG4:=LONG4, ML0=>ML428, ML1=>ML429, ML2=>ML430, ML3=>ML431);
108: DIST(LONG4:=LONG4, ML0=>ML432, ML1=>ML433, ML2=>ML434, ML3=>ML435);
109: DIST(LONG4:=LONG4, ML0=>ML436, ML1=>ML437, ML2=>ML438, ML3=>ML439);
110: DIST(LONG4:=LONG4, ML0=>ML440, ML1=>ML441, ML2=>ML442, ML3=>ML443);
111: DIST(LONG4:=LONG4, ML0=>ML444, ML1=>ML445, ML2=>ML446, ML3=>ML447);
112: DIST(LONG4:=LONG4, ML0=>ML448, ML1=>ML449, ML2=>ML450, ML3=>ML451);
113: DIST(LONG4:=LONG4, ML0=>ML452, ML1=>ML453, ML2=>ML454, ML3=>ML455);
114: DIST(LONG4:=LONG4, ML0=>ML456, ML1=>ML457, ML2=>ML458, ML3=>ML459);
115: DIST(LONG4:=LONG4, ML0=>ML460, ML1=>ML461, ML2=>ML462, ML3=>ML463);
116: DIST(LONG4:=LONG4, ML0=>ML464, ML1=>ML465, ML2=>ML466, ML3=>ML467);
117: DIST(LONG4:=LONG4, ML0=>ML468, ML1=>ML469, ML2=>ML470, ML3=>ML471);
118: DIST(LONG4:=LONG4, ML0=>ML472, ML1=>ML473, ML2=>ML474, ML3=>ML475);
119: DIST(LONG4:=LONG4, ML0=>ML476, ML1=>ML477, ML2=>ML478, ML3=>ML479);
120: DIST(LONG4:=LONG4, ML0=>ML480, ML1=>ML481, ML2=>ML482, ML3=>ML483);
121: DIST(LONG4:=LONG4, ML0=>ML484, ML1=>ML485, ML2=>ML486, ML3=>ML487);
122: DIST(LONG4:=LONG4, ML0=>ML488, ML1=>ML489, ML2=>ML490, ML3=>ML491);
123: DIST(LONG4:=LONG4, ML0=>ML492, ML1=>ML493, ML2=>ML494, ML3=>ML495);
124: DIST(LONG4:=LONG4, ML0=>ML496, ML1=>ML497, ML2=>ML498, ML3=>ML499);
125: DIST(LONG4:=LONG4, ML0=>ML500, ML1=>ML501, ML2=>ML502, ML3=>ML503);
126: DIST(LONG4:=LONG4, ML0=>ML504, ML1=>ML505, ML2=>ML506, ML3=>ML507);
127: DIST(LONG4:=LONG4, ML0=>ML508, ML1=>ML509, ML2=>ML510, ML3=>ML511);
128: DIST(LONG4:=LONG4, ML0=>ML512, ML1=>ML513, ML2=>ML514, ML3=>ML515);
129: DIST(LONG4:=LONG4, ML0=>ML516, ML1=>ML517, ML2=>ML518, ML3=>ML519);
130: DIST(LONG4:=LONG4, ML0=>ML520, ML1=>ML521, ML2=>ML522, ML3=>ML523);
131: DIST(LONG4:=LONG4, ML0=>ML524, ML1=>ML525, ML2=>ML526, ML3=>ML527);
132: DIST(LONG4:=LONG4, ML0=>ML528, ML1=>ML529, ML2=>ML530, ML3=>ML531);
133: DIST(LONG4:=LONG4, ML0=>ML532, ML1=>ML533, ML2=>ML534, ML3=>ML535);
134: DIST(LONG4:=LONG4, ML0=>ML536, ML1=>ML537, ML2=>ML538, ML3=>ML539);
135: DIST(LONG4:=LONG4, ML0=>ML540, ML1=>ML541, ML2=>ML542, ML3=>ML543);
136: DIST(LONG4:=LONG4, ML0=>ML544, ML1=>ML545, ML2=>ML546, ML3=>ML547);
137: DIST(LONG4:=LONG4, ML0=>ML548, ML1=>ML549, ML2=>ML550, ML3=>ML551);
138: DIST(LONG4:=LONG4, ML0=>ML552, ML1=>ML553, ML2=>ML554, ML3=>ML555);
139: DIST(LONG4:=LONG4, ML0=>ML556, ML1=>ML557, ML2=>ML558, ML3=>ML559);
140: DIST(LONG4:=LONG4, ML0=>ML560, ML1=>ML561, ML2=>ML562, ML3=>ML563);
141: DIST(LONG4:=LONG4, ML0=>ML564, ML1=>ML565, ML2=>ML566, ML3=>ML567);
142: DIST(LONG4:=LONG4, ML0=>ML568, ML1=>ML569, ML2=>ML570, ML3=>ML571);
143: DIST(LONG4:=LONG4, ML0=>ML572, ML1=>ML573, ML2=>ML574, ML3=>ML575);
144: DIST(LONG4:=LONG4, ML0=>ML576, ML1=>ML577, ML2=>ML578, ML3=>ML579);
145: DIST(LONG4:=LONG4, ML0=>ML580, ML1=>ML581, ML2=>ML582, ML3=>ML583);
146: DIST(LONG4:=LONG4, ML0=>ML584, ML1=>ML585, ML2=>ML586, ML3=>ML587);
147: DIST(LONG4:=LONG4, ML0=>ML588, ML1=>ML589, ML2=>ML590, ML3=>ML591);
148: DIST(LONG4:=LONG4, ML0=>ML592, ML1=>ML593, ML2=>ML594, ML3=>ML595);
149: DIST(LONG4:=LONG4, ML0=>ML596, ML1=>ML597, ML2=>ML598, ML3=>ML599);
150: DIST(LONG4:=LONG4, ML0=>ML600, ML1=>ML601, ML2=>ML602, ML3=>ML603);
151: DIST(LONG4:=LONG4, ML0=>ML604, ML1=>ML605, ML2=>ML606, ML3=>ML607);
152: DIST(LONG4:=LONG4, ML0=>ML608, ML1=>ML609, ML2=>ML610, ML3=>ML611);
153: DIST(LONG4:=LONG4, ML0=>ML612, ML1=>ML613, ML2=>ML614, ML3=>ML615);
154: DIST(LONG4:=LONG4, ML0=>ML616, ML1=>ML617, ML2=>ML618, ML3=>ML619);
155: DIST(LONG4:=LONG4, ML0=>ML620, ML1=>ML621, ML2=>ML622, ML3=>ML623);
156: DIST(LONG4:=LONG4, ML0=>ML624, ML1=>ML625, ML2=>ML626, ML3=>ML627);
157: DIST(LONG4:=LONG4, ML0=>ML628, ML1=>ML629, ML2=>ML630, ML3=>ML631);
158: DIST(LONG4:=LONG4, ML0=>ML632, ML1=>ML633, ML2=>ML634, ML3=>ML635);
159: DIST(LONG4:=LONG4, ML0=>ML636, ML1=>ML637, ML2=>ML638, ML3=>ML639);
160: DIST(LONG4:=LONG4, ML0=>ML640, ML1=>ML641, ML2=>ML642, ML3=>ML643);
161: DIST(LONG4:=LONG4, ML0=>ML644, ML1=>ML645, ML2=>ML646, ML3=>ML647);
162: DIST(LONG4:=LONG4, ML0=>ML648, ML1=>ML649, ML2=>ML650, ML3=>ML651);
163: DIST(LONG4:=LONG4, ML0=>ML652, ML1=>ML653, ML2=>ML654, ML3=>ML655);
164: DIST(LONG4:=LONG4, ML0=>ML656, ML1=>ML657, ML2=>ML658, ML3=>ML659);
165: DIST(LONG4:=LONG4, ML0=>ML660, ML1=>ML661, ML2=>ML662, ML3=>ML663);
166: DIST(LONG4:=LONG4, ML0=>ML664, ML1=>ML665, ML2=>ML666, ML3=>ML667);
167: DIST(LONG4:=LONG4, ML0=>ML668, ML1=>ML669, ML2=>ML670, ML3=>ML671);
168: DIST(LONG4:=LONG4, ML0=>ML672, ML1=>ML673, ML2=>ML674, ML3=>ML675);
169: DIST(LONG4:=LONG4, ML0=>ML676, ML1=>ML677, ML2=>ML678, ML3=>ML679);
170: DIST(LONG4:=LONG4, ML0=>ML680, ML1=>ML681, ML2=>ML682, ML3=>ML683);
171: DIST(LONG4:=LONG4, ML0=>ML684, ML1=>ML685, ML2=>ML686, ML3=>ML687);
172: DIST(LONG4:=LONG4, ML0=>ML688, ML1=>ML689, ML2=>ML690, ML3=>ML691);
173: DIST(LONG4:=LONG4, ML0=>ML692, ML1=>ML693, ML2=>ML694, ML3=>ML695);
174: DIST(LONG4:=LONG4, ML0=>ML696, ML1=>ML697, ML2=>ML698, ML3=>ML699);
175: DIST(LONG4:=LONG4, ML0=>ML700, ML1=>ML701, ML2=>ML702, ML3=>ML703);
176: DIST(LONG4:=LONG4, ML0=>ML704, ML1=>ML705, ML2=>ML706, ML3=>ML707);
177: DIST(LONG4:=LONG4, ML0=>ML708, ML1=>ML709, ML2=>ML710, ML3=>ML711);
178: DIST(LONG4:=LONG4, ML0=>ML712, ML1=>ML713, ML2=>ML714, ML3=>ML715);
179: DIST(LONG4:=LONG4, ML0=>ML716, ML1=>ML717, ML2=>ML718, ML3=>ML719);
180: DIST(LONG4:=LONG4, ML0=>ML720, ML1=>ML721, ML2=>ML722, ML3=>ML723);
181: DIST(LONG4:=LONG4, ML0=>ML724, ML1=>ML725, ML2=>ML726, ML3=>ML727);
182: DIST(LONG4:=LONG4, ML0=>ML728, ML1=>ML729, ML2=>ML730, ML3=>ML731);
183: DIST(LONG4:=LONG4, ML0=>ML732, ML1=>ML733, ML2=>ML734, ML3=>ML735);
184: DIST(LONG4:=LONG4, ML0=>ML736, ML1=>ML737, ML2=>ML738, ML3=>ML739);
185: DIST(LONG4:=LONG4, ML0=>ML740, ML1=>ML741, ML2=>ML742, ML3=>ML743);
186: DIST(LONG4:=LONG4, ML0=>ML744, ML1=>ML745, ML2=>ML746, ML3=>ML747);
187: DIST(LONG4:=LONG4, ML0=>ML748, ML1=>ML749, ML2=>ML750, ML3=>ML751);
188: DIST(LONG4:=LONG4, ML0=>ML752, ML1=>ML753, ML2=>ML754, ML3=>ML755);
189: DIST(LONG4:=LONG4, ML0=>ML756, ML1=>ML757, ML2=>ML758, ML3=>ML759);
190: DIST(LONG4:=LONG4, ML0=>ML760, ML1=>ML761, ML2=>ML762, ML3=>ML763);
191: DIST(LONG4:=LONG4, ML0=>ML764, ML1=>ML765, ML2=>ML766, ML3=>ML767);
192: DIST(LONG4:=LONG4, ML0=>ML768, ML1=>ML769, ML2=>ML770, ML3=>ML771);
193: DIST(LONG4:=LONG4, ML0=>ML772, ML1=>ML773, ML2=>ML774, ML3=>ML775);
194: DIST(LONG4:=LONG4, ML0=>ML776, ML1=>ML777, ML2=>ML778, ML3=>ML779);
195: DIST(LONG4:=LONG4, ML0=>ML780, ML1=>ML781, ML2=>ML782, ML3=>ML783);
196: DIST(LONG4:=LONG4, ML0=>ML784, ML1=>ML785, ML2=>ML786, ML3=>ML787);
197: DIST(LONG4:=LONG4, ML0=>ML788, ML1=>ML789, ML2=>ML790, ML3=>ML791);
198: DIST(LONG4:=LONG4, ML0=>ML792, ML1=>ML793, ML2=>ML794, ML3=>ML795);
199: DIST(LONG4:=LONG4, ML0=>ML796, ML1=>ML797, ML2=>ML798, ML3=>ML799);
200: DIST(LONG4:=LONG4, ML0=>ML800, ML1=>ML801, ML2=>ML802, ML3=>ML803);
201: DIST(LONG4:=LONG4, ML0=>ML804, ML1=>ML805, ML2=>ML806, ML3=>ML807);
202: DIST(LONG4:=LONG4, ML0=>ML808, ML1=>ML809, ML2=>ML810, ML3=>ML811);
203: DIST(LONG4:=LONG4, ML0=>ML812, ML1=>ML813, ML2=>ML814, ML3=>ML815);
204: DIST(LONG4:=LONG4, ML0=>ML816, ML1=>ML817, ML2=>ML818, ML3=>ML819);
205: DIST(LONG4:=LONG4, ML0=>ML820, ML1=>ML821, ML2=>ML822, ML3=>ML823);
206: DIST(LONG4:=LONG4, ML0=>ML824, ML1=>ML825, ML2=>ML826, ML3=>ML827);
207: DIST(LONG4:=LONG4, ML0=>ML828, ML1=>ML829, ML2=>ML830, ML3=>ML831);
208: DIST(LONG4:=LONG4, ML0=>ML832, ML1=>ML833, ML2=>ML834, ML3=>ML835);
209: DIST(LONG4:=LONG4, ML0=>ML836, ML1=>ML837, ML2=>ML838, ML3=>ML839);
210: DIST(LONG4:=LONG4, ML0=>ML840, ML1=>ML841, ML2=>ML842, ML3=>ML843);
211: DIST(LONG4:=LONG4, ML0=>ML844, ML1=>ML845, ML2=>ML846, ML3=>ML847);
212: DIST(LONG4:=LONG4, ML0=>ML848, ML1=>ML849, ML2=>ML850, ML3=>ML851);
213: DIST(LONG4:=LONG4, ML0=>ML852, ML1=>ML853, ML2=>ML854, ML3=>ML855);
214: DIST(LONG4:=LONG4, ML0=>ML856, ML1=>ML857, ML2=>ML858, ML3=>ML859);
215: DIST(LONG4:=LONG4, ML0=>ML860, ML1=>ML861, ML2=>ML862, ML3=>ML863);
216: DIST(LONG4:=LONG4, ML0=>ML864, ML1=>ML865, ML2=>ML866, ML3=>ML867);
217: DIST(LONG4:=LONG4, ML0=>ML868, ML1=>ML869, ML2=>ML870, ML3=>ML871);
218: DIST(LONG4:=LONG4, ML0=>ML872, ML1=>ML873, ML2=>ML874, ML3=>ML875);
219: DIST(LONG4:=LONG4, ML0=>ML876, ML1=>ML877, ML2=>ML878, ML3=>ML879);
220: DIST(LONG4:=LONG4, ML0=>ML880, ML1=>ML881, ML2=>ML882, ML3=>ML883);
221: DIST(LONG4:=LONG4, ML0=>ML884, ML1=>ML885, ML2=>ML886, ML3=>ML887);
222: DIST(LONG4:=LONG4, ML0=>ML888, ML1=>ML889, ML2=>ML890, ML3=>ML891);
223: DIST(LONG4:=LONG4, ML0=>ML892, ML1=>ML893, ML2=>ML894, ML3=>ML895);
224: DIST(LONG4:=LONG4, ML0=>ML896, ML1=>ML897, ML2=>ML898, ML3=>ML899);
225: DIST(LONG4:=LONG4, ML0=>ML900, ML1=>ML901, ML2=>ML902, ML3=>ML903);
226: DIST(LONG4:=LONG4, ML0=>ML904, ML1=>ML905, ML2=>ML906, ML3=>ML907);
227: DIST(LONG4:=LONG4, ML0=>ML908, ML1=>ML909, ML2=>ML910, ML3=>ML911);
228: DIST(LONG4:=LONG4, ML0=>ML912, ML1=>ML913, ML2=>ML914, ML3=>ML915);
229: DIST(LONG4:=LONG4, ML0=>ML916, ML1=>ML917, ML2=>ML918, ML3=>ML919);
230: DIST(LONG4:=LONG4, ML0=>ML920, ML1=>ML921, ML2=>ML922, ML3=>ML923);
231: DIST(LONG4:=LONG4, ML0=>ML924, ML1=>ML925, ML2=>ML926, ML3=>ML927);
232: DIST(LONG4:=LONG4, ML0=>ML928, ML1=>ML929, ML2=>ML930, ML3=>ML931);
233: DIST(LONG4:=LONG4, ML0=>ML932, ML1=>ML933, ML2=>ML934, ML3=>ML935);
234: DIST(LONG4:=LONG4, ML0=>ML936, ML1=>ML937, ML2=>ML938, ML3=>ML939);
235: DIST(LONG4:=LONG4, ML0=>ML940, ML1=>ML941, ML2=>ML942, ML3=>ML943);
236: DIST(LONG4:=LONG4, ML0=>ML944, ML1=>ML945, ML2=>ML946, ML3=>ML947);
237: DIST(LONG4:=LONG4, ML0=>ML948, ML1=>ML949, ML2=>ML950, ML3=>ML951);
238: DIST(LONG4:=LONG4, ML0=>ML952, ML1=>ML953, ML2=>ML954, ML3=>ML955);
239: DIST(LONG4:=LONG4, ML0=>ML956, ML1=>ML957, ML2=>ML958, ML3=>ML959);
240: DIST(LONG4:=LONG4, ML0=>ML960, ML1=>ML961, ML2=>ML962, ML3=>ML963);
241: DIST(LONG4:=LONG4, ML0=>ML964, ML1=>ML965, ML2=>ML966, ML3=>ML967);
242: DIST(LONG4:=LONG4, ML0=>ML968, ML1=>ML969, ML2=>ML970, ML3=>ML971);
243: DIST(LONG4:=LONG4, ML0=>ML972, ML1=>ML973, ML2=>ML974, ML3=>ML975);
244: DIST(LONG4:=LONG4, ML0=>ML976, ML1=>ML977, ML2=>ML978, ML3=>ML979);
245: DIST(LONG4:=LONG4, ML0=>ML980, ML1=>ML981, ML2=>ML982, ML3=>ML983);
246: DIST(LONG4:=LONG4, ML0=>ML984, ML1=>ML985, ML2=>ML986, ML3=>ML987);
247: DIST(LONG4:=LONG4, ML0=>ML988, ML1=>ML989, ML2=>ML990, ML3=>ML991);
248: DIST(LONG4:=LONG4, ML0=>ML992, ML1=>ML993, ML2=>ML994, ML3=>ML995);
249: DIST(LONG4:=LONG4, ML0=>ML996, ML1=>ML997, ML2=>ML998, ML3=>ML999);
250: DIST(LONG4:=LONG4, ML0=>ML1000, ML1=>ML1001, ML2=>ML1002, ML3=>ML1003);
251: DIST(LONG4:=LONG4, ML0=>ML1004, ML1=>ML1005, ML2=>ML1006, ML3=>ML1007);
252: DIST(LONG4:=LONG4, ML0=>ML1008, ML1=>ML1009, ML2=>ML1010, ML3=>ML1011);
253: DIST(LONG4:=LONG4, ML0=>ML1012, ML1=>ML1013, ML2=>ML1014, ML3=>ML1015);
254: DIST(LONG4:=LONG4, ML0=>ML1016, ML1=>ML1017, ML2=>ML1018, ML3=>ML1019);
255: DIST(LONG4:=LONG4, ML0=>ML1020, ML1=>ML1021, ML2=>ML1022, ML3=>ML1023);
END_CASE;
          
END_FUNCTION_BLOCK

(* Запись сетки элемента в регистры *)
FUNCTION_BLOCK Grid2ul
  VAR_INPUT
    HGR : THandle := 0;  (* Дескриптор массива сеток *)
    PGR : TPos8 := -1;  (* Индекс сетки в массиве <HRG>[PGR] *)
    SH : TShape;  (* Фигура элемента *)
  END_VAR
  VAR_OUTPUT
    iRes : TError := E_SUCCESS;  (* Результат *)
    iLog : INT := 0;  (* Счётчик строк протокола *)
  END_VAR
  VAR
    msg : STRING := '0';  (* Сообщение в протокол *)
    _SetLong4 : SetLong4;  (* Запись 4-х ULINT в массив ML[0..1023] *)
  END_VAR

            VAR
  m4,n4,idx   : INT;       (* счётчики слов        *)  
  i,j,k       : INT;       (* индексы узлов сетки  *)  
  w: ARRAY[0..3] of INT;   (* буфер 2-байтных слов *)
  l: ARRAY[0..3] of ULINT; (* буфер 4-байтных слов *)
END_VAR

(* Установка начальных значений *)
iLog:=0;
iRes := E_FAIL;
m4:=0; n4:=0; idx:=0;

(* Запись значений температуры сетки в регистры *)
FOR k := 0 TO SH.Kn[2]-1 DO 
  FOR j := 0 TO SH.Kn[1]-1 DO 
    FOR i := 0 TO SH.Kn[0]-1 DO 

      w[m4]:=var_v(
        get_var( HGR, PGR, 
          knoff(SH.Kn[0], SH.Kn[1], SH.Kn[2], i, j, k)
        )
      );
      
      if (iLog<4096) then  
        if (len(msg)=0) then msg := MakeMsg(' =!=> '); end_if;
        msg := MakeMsg(msg, INT_TO_STRING(w[m4]), ' ');
        if (mod((iLog+1),64)=0) then msg:=LogMsg(MakeMsg(msg)); end_if;
        iLog:=iLog+1;
      end_if;
      
      m4 := m4+1;
      if (mod(m4, 4)=0) then 
        m4 := 0;
        
        (*
        if (iLog<64) then  
          if (len(msg)=0) then msg := MakeMsg(' => '); end_if;
          msg := MakeMsg(msg, '[', INT_TO_STRING(w[0]), ',');
          msg := MakeMsg(msg,  '', INT_TO_STRING(w[1]), ',');
          msg := MakeMsg(msg,  '', INT_TO_STRING(w[2]), ',');
          msg := MakeMsg(msg,  '', INT_TO_STRING(w[3]), ']');
        end_if;
        *)
        
        l[n4] := int4ul(w[0], w[1], w[2], w[3]); 
        
        n4 := n4+1;
        if (mod(n4, 4)=0) then 
          n4 := 0;
        
          (*if (iLog<64) then msg:=LogMsg(MakeMsg(msg,';')); iLog:=iLog+1; end_if;*)
          
          _SetLong4(I:=idx, LONG4:=l); idx := idx+1;
        end_if;
        
      end_if;
      
    END_FOR; 
  END_FOR; 
END_FOR;

if (len(msg)>0) then msg:=LogMsg(MakeMsg(msg)); end_if;

(* Установка результата *)
if (mod(m4,4)<>0) or (mod(n4,4)<>0) then 
      iRes:=E_INDEX;    (* ошибка индекса    *)
else  iRes:=E_SUCCESS;  (* выполнено успешно *)
end_if; 

          
END_FUNCTION_BLOCK

(* Выкладка состояния элемента *)
FUNCTION_BLOCK DistCond
  VAR_OUTPUT
    MD0 : UDINT := 0;
    MD1 : UDINT := 0;
    MD2 : UDINT := 0;
    MD3 : UDINT := 0;
    MD4 : UDINT := 0;
  END_VAR
  VAR_INPUT
    COND : TCond;  (* Объект "Состояние элемента" *)
  END_VAR

            MD0 := UINT_TO_UDINT(COND.ID)*65536 + INT_TO_UDINT(COND.Tmid);

MD1 := INT_TO_UDINT(COND.Tmin.A[0])*65536 + INT_TO_UDINT(COND.Tmin.A[1]);
MD2 := INT_TO_UDINT(COND.Tmin.A[2])*65536 + INT_TO_UDINT(COND.Tmin.V);

MD3 := INT_TO_UDINT(COND.Tmax.A[0])*65536 + INT_TO_UDINT(COND.Tmax.A[1]);
MD4 := INT_TO_UDINT(COND.Tmax.A[2])*65536 + INT_TO_UDINT(COND.Tmax.V);

          
END_FUNCTION_BLOCK

(* Чтение состояния элемента из регистров *)
FUNCTION_BLOCK SetCond
  VAR_EXTERNAL
    MW1000 : UINT;
    MW1001 : UINT;
    MW1002 : UINT;
    MW1003 : UINT;
    MW1004 : UINT;
    MW1005 : UINT;
    MW1006 : UINT;
    MW1007 : UINT;
    MW1008 : UINT;
    MW1009 : UINT;
    MD500 : UDINT;
    MD501 : UDINT;
    MD502 : UDINT;
    MD503 : UDINT;
    MD504 : UDINT;
    MD505 : UDINT;
    MD506 : UDINT;
    MD507 : UDINT;
    MD508 : UDINT;
    MD509 : UDINT;
    MD510 : UDINT;
    MD511 : UDINT;
    MD512 : UDINT;
    MD513 : UDINT;
    MD514 : UDINT;
    MD515 : UDINT;
    MD516 : UDINT;
    MD517 : UDINT;
    MD518 : UDINT;
    MD519 : UDINT;
    MD520 : UDINT;
    MD521 : UDINT;
    MD522 : UDINT;
    MD523 : UDINT;
    MD524 : UDINT;
    MD525 : UDINT;
    MD526 : UDINT;
    MD527 : UDINT;
    MD528 : UDINT;
    MD529 : UDINT;
    MD530 : UDINT;
    MD531 : UDINT;
    MD532 : UDINT;
    MD533 : UDINT;
    MD534 : UDINT;
    MD535 : UDINT;
    MD536 : UDINT;
    MD537 : UDINT;
    MD538 : UDINT;
    MD539 : UDINT;
    MD540 : UDINT;
    MD541 : UDINT;
    MD542 : UDINT;
    MD543 : UDINT;
    MD544 : UDINT;
    MD545 : UDINT;
    MD546 : UDINT;
    MD547 : UDINT;
    MD548 : UDINT;
    MD549 : UDINT;
    MD550 : UDINT;
    MD551 : UDINT;
    MD552 : UDINT;
    MD553 : UDINT;
    MD554 : UDINT;
    MD555 : UDINT;
    MD556 : UDINT;
    MD557 : UDINT;
    MD558 : UDINT;
    MD559 : UDINT;
    MD560 : UDINT;
    MD561 : UDINT;
    MD562 : UDINT;
    MD563 : UDINT;
    MD564 : UDINT;
    MD565 : UDINT;
    MD566 : UDINT;
    MD567 : UDINT;
    MD568 : UDINT;
    MD569 : UDINT;
    MD570 : UDINT;
    MD571 : UDINT;
    MD572 : UDINT;
    MD573 : UDINT;
    MD574 : UDINT;
    MD575 : UDINT;
    MD576 : UDINT;
    MD577 : UDINT;
    MD578 : UDINT;
    MD579 : UDINT;
    MD580 : UDINT;
    MD581 : UDINT;
    MD582 : UDINT;
    MD583 : UDINT;
    MD584 : UDINT;
    MD585 : UDINT;
    MD586 : UDINT;
    MD587 : UDINT;
    MD588 : UDINT;
    MD589 : UDINT;
    MD590 : UDINT;
    MD591 : UDINT;
    MD592 : UDINT;
    MD593 : UDINT;
    MD594 : UDINT;
    MD595 : UDINT;
    MD596 : UDINT;
    MD597 : UDINT;
    MD598 : UDINT;
    MD599 : UDINT;
    MD600 : UDINT;
    MD601 : UDINT;
    MD602 : UDINT;
    MD603 : UDINT;
    MD604 : UDINT;
    MD605 : UDINT;
    MD606 : UDINT;
    MD607 : UDINT;
    MD608 : UDINT;
    MD609 : UDINT;
    MD610 : UDINT;
    MD611 : UDINT;
    MD612 : UDINT;
    MD613 : UDINT;
    MD614 : UDINT;
    MD615 : UDINT;
    MD616 : UDINT;
    MD617 : UDINT;
    MD618 : UDINT;
    MD619 : UDINT;
    MD620 : UDINT;
    MD621 : UDINT;
    MD622 : UDINT;
    MD623 : UDINT;
    MD624 : UDINT;
    MD625 : UDINT;
    MD626 : UDINT;
    MD627 : UDINT;
    MD628 : UDINT;
    MD629 : UDINT;
    MD630 : UDINT;
    MD631 : UDINT;
    MD632 : UDINT;
    MD633 : UDINT;
    MD634 : UDINT;
    MD635 : UDINT;
    MD636 : UDINT;
    MD637 : UDINT;
    MD638 : UDINT;
    MD639 : UDINT;
    MD640 : UDINT;
    MD641 : UDINT;
    MD642 : UDINT;
    MD643 : UDINT;
    MD644 : UDINT;
    MD645 : UDINT;
    MD646 : UDINT;
    MD647 : UDINT;
    MD648 : UDINT;
    MD649 : UDINT;
    MD650 : UDINT;
    MD651 : UDINT;
    MD652 : UDINT;
    MD653 : UDINT;
    MD654 : UDINT;
    MD655 : UDINT;
    MD656 : UDINT;
    MD657 : UDINT;
    MD658 : UDINT;
    MD659 : UDINT;
    MD660 : UDINT;
    MD661 : UDINT;
    MD662 : UDINT;
    MD663 : UDINT;
    MD664 : UDINT;
    MD665 : UDINT;
    MD666 : UDINT;
    MD667 : UDINT;
    MD668 : UDINT;
    MD669 : UDINT;
    MD670 : UDINT;
    MD671 : UDINT;
    MD672 : UDINT;
    MD673 : UDINT;
    MD674 : UDINT;
    MD675 : UDINT;
    MD676 : UDINT;
    MD677 : UDINT;
    MD678 : UDINT;
    MD679 : UDINT;
    MD680 : UDINT;
    MD681 : UDINT;
    MD682 : UDINT;
    MD683 : UDINT;
    MD684 : UDINT;
    MD685 : UDINT;
    MD686 : UDINT;
    MD687 : UDINT;
    MD688 : UDINT;
    MD689 : UDINT;
    MD690 : UDINT;
    MD691 : UDINT;
    MD692 : UDINT;
    MD693 : UDINT;
    MD694 : UDINT;
    MD695 : UDINT;
    MD696 : UDINT;
    MD697 : UDINT;
    MD698 : UDINT;
    MD699 : UDINT;
    MD700 : UDINT;
    MD701 : UDINT;
    MD702 : UDINT;
    MD703 : UDINT;
    MD704 : UDINT;
    MD705 : UDINT;
    MD706 : UDINT;
    MD707 : UDINT;
    MD708 : UDINT;
    MD709 : UDINT;
    MD710 : UDINT;
    MD711 : UDINT;
    MD712 : UDINT;
    MD713 : UDINT;
    MD714 : UDINT;
    MD715 : UDINT;
    MD716 : UDINT;
    MD717 : UDINT;
    MD718 : UDINT;
    MD719 : UDINT;
    MD720 : UDINT;
    MD721 : UDINT;
    MD722 : UDINT;
    MD723 : UDINT;
    MD724 : UDINT;
    MD725 : UDINT;
    MD726 : UDINT;
    MD727 : UDINT;
    MD728 : UDINT;
    MD729 : UDINT;
    MD730 : UDINT;
    MD731 : UDINT;
    MD732 : UDINT;
    MD733 : UDINT;
    MD734 : UDINT;
    MD735 : UDINT;
    MD736 : UDINT;
    MD737 : UDINT;
    MD738 : UDINT;
    MD739 : UDINT;
    MD740 : UDINT;
    MD741 : UDINT;
    MD742 : UDINT;
    MD743 : UDINT;
    MD744 : UDINT;
    MD745 : UDINT;
    MD746 : UDINT;
    MD747 : UDINT;
    MD748 : UDINT;
    MD749 : UDINT;
    MD750 : UDINT;
    MD751 : UDINT;
    MD752 : UDINT;
    MD753 : UDINT;
    MD754 : UDINT;
    MD755 : UDINT;
    MD756 : UDINT;
    MD757 : UDINT;
    MD758 : UDINT;
    MD759 : UDINT;
    MD760 : UDINT;
    MD761 : UDINT;
    MD762 : UDINT;
    MD763 : UDINT;
    MD764 : UDINT;
    MD765 : UDINT;
    MD766 : UDINT;
    MD767 : UDINT;
    MD768 : UDINT;
    MD769 : UDINT;
    MD770 : UDINT;
    MD771 : UDINT;
    MD772 : UDINT;
    MD773 : UDINT;
    MD774 : UDINT;
    MD775 : UDINT;
    MD776 : UDINT;
    MD777 : UDINT;
    MD778 : UDINT;
    MD779 : UDINT;
    MD780 : UDINT;
    MD781 : UDINT;
    MD782 : UDINT;
    MD783 : UDINT;
    MD784 : UDINT;
    MD785 : UDINT;
    MD786 : UDINT;
    MD787 : UDINT;
    MD788 : UDINT;
    MD789 : UDINT;
    MD790 : UDINT;
    MD791 : UDINT;
    MD792 : UDINT;
    MD793 : UDINT;
    MD794 : UDINT;
    MD795 : UDINT;
    MD796 : UDINT;
    MD797 : UDINT;
    MD798 : UDINT;
    MD799 : UDINT;
    MD800 : UDINT;
    MD801 : UDINT;
    MD802 : UDINT;
    MD803 : UDINT;
    MD804 : UDINT;
    MD805 : UDINT;
    MD806 : UDINT;
    MD807 : UDINT;
    MD808 : UDINT;
    MD809 : UDINT;
    MD810 : UDINT;
    MD811 : UDINT;
    MD812 : UDINT;
    MD813 : UDINT;
    MD814 : UDINT;
    MD815 : UDINT;
    MD816 : UDINT;
    MD817 : UDINT;
    MD818 : UDINT;
    MD819 : UDINT;
    MD820 : UDINT;
    MD821 : UDINT;
    MD822 : UDINT;
    MD823 : UDINT;
    MD824 : UDINT;
    MD825 : UDINT;
    MD826 : UDINT;
    MD827 : UDINT;
    MD828 : UDINT;
    MD829 : UDINT;
    MD830 : UDINT;
    MD831 : UDINT;
    MD832 : UDINT;
    MD833 : UDINT;
    MD834 : UDINT;
    MD835 : UDINT;
    MD836 : UDINT;
    MD837 : UDINT;
    MD838 : UDINT;
    MD839 : UDINT;
    MD840 : UDINT;
    MD841 : UDINT;
    MD842 : UDINT;
    MD843 : UDINT;
    MD844 : UDINT;
    MD845 : UDINT;
    MD846 : UDINT;
    MD847 : UDINT;
    MD848 : UDINT;
    MD849 : UDINT;
    MD850 : UDINT;
    MD851 : UDINT;
    MD852 : UDINT;
    MD853 : UDINT;
    MD854 : UDINT;
    MD855 : UDINT;
    MD856 : UDINT;
    MD857 : UDINT;
    MD858 : UDINT;
    MD859 : UDINT;
    MD860 : UDINT;
    MD861 : UDINT;
    MD862 : UDINT;
    MD863 : UDINT;
    MD864 : UDINT;
    MD865 : UDINT;
    MD866 : UDINT;
    MD867 : UDINT;
    MD868 : UDINT;
    MD869 : UDINT;
    MD870 : UDINT;
    MD871 : UDINT;
    MD872 : UDINT;
    MD873 : UDINT;
    MD874 : UDINT;
    MD875 : UDINT;
    MD876 : UDINT;
    MD877 : UDINT;
    MD878 : UDINT;
    MD879 : UDINT;
    MD880 : UDINT;
    MD881 : UDINT;
    MD882 : UDINT;
    MD883 : UDINT;
    MD884 : UDINT;
    MD885 : UDINT;
    MD886 : UDINT;
    MD887 : UDINT;
    MD888 : UDINT;
    MD889 : UDINT;
    MD890 : UDINT;
    MD891 : UDINT;
    MD892 : UDINT;
    MD893 : UDINT;
    MD894 : UDINT;
    MD895 : UDINT;
    MD896 : UDINT;
    MD897 : UDINT;
    MD898 : UDINT;
    MD899 : UDINT;
    MD900 : UDINT;
    MD901 : UDINT;
    MD902 : UDINT;
    MD903 : UDINT;
    MD904 : UDINT;
    MD905 : UDINT;
    MD906 : UDINT;
    MD907 : UDINT;
    MD908 : UDINT;
    MD909 : UDINT;
    MD910 : UDINT;
    MD911 : UDINT;
    MD912 : UDINT;
    MD913 : UDINT;
    MD914 : UDINT;
    MD915 : UDINT;
    MD916 : UDINT;
    MD917 : UDINT;
    MD918 : UDINT;
    MD919 : UDINT;
    MD920 : UDINT;
    MD921 : UDINT;
    MD922 : UDINT;
    MD923 : UDINT;
    MD924 : UDINT;
    MD925 : UDINT;
    MD926 : UDINT;
    MD927 : UDINT;
    MD928 : UDINT;
    MD929 : UDINT;
    MD930 : UDINT;
    MD931 : UDINT;
    MD932 : UDINT;
    MD933 : UDINT;
    MD934 : UDINT;
    MD935 : UDINT;
    MD936 : UDINT;
    MD937 : UDINT;
    MD938 : UDINT;
    MD939 : UDINT;
    MD940 : UDINT;
    MD941 : UDINT;
    MD942 : UDINT;
    MD943 : UDINT;
    MD944 : UDINT;
    MD945 : UDINT;
    MD946 : UDINT;
    MD947 : UDINT;
    MD948 : UDINT;
    MD949 : UDINT;
    MD950 : UDINT;
    MD951 : UDINT;
    MD952 : UDINT;
    MD953 : UDINT;
    MD954 : UDINT;
    MD955 : UDINT;
    MD956 : UDINT;
    MD957 : UDINT;
    MD958 : UDINT;
    MD959 : UDINT;
    MD960 : UDINT;
    MD961 : UDINT;
    MD962 : UDINT;
    MD963 : UDINT;
    MD964 : UDINT;
    MD965 : UDINT;
    MD966 : UDINT;
    MD967 : UDINT;
    MD968 : UDINT;
    MD969 : UDINT;
    MD970 : UDINT;
    MD971 : UDINT;
    MD972 : UDINT;
    MD973 : UDINT;
    MD974 : UDINT;
    MD975 : UDINT;
    MD976 : UDINT;
    MD977 : UDINT;
    MD978 : UDINT;
    MD979 : UDINT;
    MD980 : UDINT;
    MD981 : UDINT;
    MD982 : UDINT;
    MD983 : UDINT;
    MD984 : UDINT;
    MD985 : UDINT;
    MD986 : UDINT;
    MD987 : UDINT;
    MD988 : UDINT;
    MD989 : UDINT;
    MD990 : UDINT;
    MD991 : UDINT;
    MD992 : UDINT;
    MD993 : UDINT;
    MD994 : UDINT;
    MD995 : UDINT;
    MD996 : UDINT;
    MD997 : UDINT;
    MD998 : UDINT;
    MD999 : UDINT;
  END_VAR
  VAR_INPUT
    I : UINT := 0;
    COND : TCond;
  END_VAR
  VAR
    DIST : DistCond;
    msg : STRING := '';
  END_VAR

            CASE i OF
0  : DIST(COND:=COND,MD0=>MD500,MD1=>MD501,MD2=>MD502,MD3=>MD503,MD4=>MD504);
1  : DIST(COND:=COND,MD0=>MD505,MD1=>MD506,MD2=>MD507,MD3=>MD508,MD4=>MD509);
2  : DIST(COND:=COND,MD0=>MD510,MD1=>MD511,MD2=>MD512,MD3=>MD513,MD4=>MD514);
3  : DIST(COND:=COND,MD0=>MD515,MD1=>MD516,MD2=>MD517,MD3=>MD518,MD4=>MD519);
4  : DIST(COND:=COND,MD0=>MD520,MD1=>MD521,MD2=>MD522,MD3=>MD523,MD4=>MD524);
5  : DIST(COND:=COND,MD0=>MD525,MD1=>MD526,MD2=>MD527,MD3=>MD528,MD4=>MD529);
6  : DIST(COND:=COND,MD0=>MD530,MD1=>MD531,MD2=>MD532,MD3=>MD533,MD4=>MD534);
7  : DIST(COND:=COND,MD0=>MD535,MD1=>MD536,MD2=>MD537,MD3=>MD538,MD4=>MD539);
8  : DIST(COND:=COND,MD0=>MD540,MD1=>MD541,MD2=>MD542,MD3=>MD543,MD4=>MD544);
9  : DIST(COND:=COND,MD0=>MD545,MD1=>MD546,MD2=>MD547,MD3=>MD548,MD4=>MD549);

10 : DIST(COND:=COND,MD0=>MD550,MD1=>MD551,MD2=>MD552,MD3=>MD553,MD4=>MD554);
11 : DIST(COND:=COND,MD0=>MD555,MD1=>MD556,MD2=>MD557,MD3=>MD558,MD4=>MD559);
12 : DIST(COND:=COND,MD0=>MD560,MD1=>MD561,MD2=>MD562,MD3=>MD563,MD4=>MD564);
13 : DIST(COND:=COND,MD0=>MD565,MD1=>MD566,MD2=>MD567,MD3=>MD568,MD4=>MD569);
14 : DIST(COND:=COND,MD0=>MD570,MD1=>MD571,MD2=>MD572,MD3=>MD573,MD4=>MD574);
15 : DIST(COND:=COND,MD0=>MD575,MD1=>MD576,MD2=>MD577,MD3=>MD578,MD4=>MD579);
16 : DIST(COND:=COND,MD0=>MD580,MD1=>MD581,MD2=>MD582,MD3=>MD583,MD4=>MD584);
17 : DIST(COND:=COND,MD0=>MD585,MD1=>MD586,MD2=>MD587,MD3=>MD588,MD4=>MD589);
18 : DIST(COND:=COND,MD0=>MD590,MD1=>MD591,MD2=>MD592,MD3=>MD593,MD4=>MD594);
19 : DIST(COND:=COND,MD0=>MD595,MD1=>MD596,MD2=>MD597,MD3=>MD598,MD4=>MD599);

20 : DIST(COND:=COND,MD0=>MD600,MD1=>MD601,MD2=>MD602,MD3=>MD603,MD4=>MD604);
21 : DIST(COND:=COND,MD0=>MD605,MD1=>MD606,MD2=>MD607,MD3=>MD608,MD4=>MD609);
22 : DIST(COND:=COND,MD0=>MD610,MD1=>MD611,MD2=>MD612,MD3=>MD613,MD4=>MD614);
23 : DIST(COND:=COND,MD0=>MD615,MD1=>MD616,MD2=>MD617,MD3=>MD618,MD4=>MD619);
24 : DIST(COND:=COND,MD0=>MD620,MD1=>MD621,MD2=>MD622,MD3=>MD623,MD4=>MD624);
25 : DIST(COND:=COND,MD0=>MD625,MD1=>MD626,MD2=>MD627,MD3=>MD628,MD4=>MD629);
26 : DIST(COND:=COND,MD0=>MD630,MD1=>MD631,MD2=>MD632,MD3=>MD633,MD4=>MD634);
27 : DIST(COND:=COND,MD0=>MD635,MD1=>MD636,MD2=>MD637,MD3=>MD638,MD4=>MD639);
28 : DIST(COND:=COND,MD0=>MD640,MD1=>MD641,MD2=>MD642,MD3=>MD643,MD4=>MD644);
29 : DIST(COND:=COND,MD0=>MD645,MD1=>MD646,MD2=>MD647,MD3=>MD648,MD4=>MD649);

30 : DIST(COND:=COND,MD0=>MD650,MD1=>MD651,MD2=>MD652,MD3=>MD653,MD4=>MD654);
31 : DIST(COND:=COND,MD0=>MD655,MD1=>MD656,MD2=>MD657,MD3=>MD658,MD4=>MD659);
32 : DIST(COND:=COND,MD0=>MD660,MD1=>MD661,MD2=>MD662,MD3=>MD663,MD4=>MD664);
33 : DIST(COND:=COND,MD0=>MD665,MD1=>MD666,MD2=>MD667,MD3=>MD668,MD4=>MD669);
34 : DIST(COND:=COND,MD0=>MD670,MD1=>MD671,MD2=>MD672,MD3=>MD673,MD4=>MD674);
35 : DIST(COND:=COND,MD0=>MD675,MD1=>MD676,MD2=>MD677,MD3=>MD678,MD4=>MD679);
36 : DIST(COND:=COND,MD0=>MD680,MD1=>MD681,MD2=>MD682,MD3=>MD683,MD4=>MD684);
37 : DIST(COND:=COND,MD0=>MD685,MD1=>MD686,MD2=>MD687,MD3=>MD688,MD4=>MD689);
38 : DIST(COND:=COND,MD0=>MD690,MD1=>MD691,MD2=>MD692,MD3=>MD693,MD4=>MD694);
39 : DIST(COND:=COND,MD0=>MD695,MD1=>MD696,MD2=>MD697,MD3=>MD698,MD4=>MD699);

40 : DIST(COND:=COND,MD0=>MD700,MD1=>MD701,MD2=>MD702,MD3=>MD703,MD4=>MD704);
41 : DIST(COND:=COND,MD0=>MD705,MD1=>MD706,MD2=>MD707,MD3=>MD708,MD4=>MD709);
42 : DIST(COND:=COND,MD0=>MD710,MD1=>MD711,MD2=>MD712,MD3=>MD713,MD4=>MD714);
43 : DIST(COND:=COND,MD0=>MD715,MD1=>MD716,MD2=>MD717,MD3=>MD718,MD4=>MD719);
44 : DIST(COND:=COND,MD0=>MD720,MD1=>MD721,MD2=>MD722,MD3=>MD723,MD4=>MD724);
45 : DIST(COND:=COND,MD0=>MD725,MD1=>MD726,MD2=>MD727,MD3=>MD728,MD4=>MD729);
46 : DIST(COND:=COND,MD0=>MD730,MD1=>MD731,MD2=>MD732,MD3=>MD733,MD4=>MD734);
47 : DIST(COND:=COND,MD0=>MD735,MD1=>MD736,MD2=>MD737,MD3=>MD738,MD4=>MD739);
48 : DIST(COND:=COND,MD0=>MD740,MD1=>MD741,MD2=>MD742,MD3=>MD743,MD4=>MD744);
49 : DIST(COND:=COND,MD0=>MD745,MD1=>MD746,MD2=>MD747,MD3=>MD748,MD4=>MD749);

50 : DIST(COND:=COND,MD0=>MD750,MD1=>MD751,MD2=>MD752,MD3=>MD753,MD4=>MD754);
51 : DIST(COND:=COND,MD0=>MD755,MD1=>MD756,MD2=>MD757,MD3=>MD758,MD4=>MD759);
52 : DIST(COND:=COND,MD0=>MD760,MD1=>MD761,MD2=>MD762,MD3=>MD763,MD4=>MD764);
53 : DIST(COND:=COND,MD0=>MD765,MD1=>MD766,MD2=>MD767,MD3=>MD768,MD4=>MD769);
(*TEST*)
(*
mw1000 := UDINT_TO_UINT(MD765/65536);
mw1001 := UDINT_TO_UINT(mod(MD765,65536));

mw1002 := UDINT_TO_UINT(MD766/65536);
mw1003 := UDINT_TO_UINT(mod(MD766,65536));
mw1004 := UDINT_TO_UINT(MD767/65536);
mw1005 := UDINT_TO_UINT(mod(MD767,65536));

mw1006 := UDINT_TO_UINT(MD768/65536);
mw1007 := UDINT_TO_UINT(mod(MD768,65536));
mw1008 := UDINT_TO_UINT(MD769/65536);
mw1009 := UDINT_TO_UINT(mod(MD769,65536));

msg := MakeMsg('= TEST2: Tmax.P(53) = [');
msg := MakeMsg(msg, INT_TO_STRING(UINT_TO_INT(mw1006)), ',');
msg := MakeMsg(msg, INT_TO_STRING(UINT_TO_INT(mw1007)), ',');
msg := MakeMsg(msg, INT_TO_STRING(UINT_TO_INT(mw1008)), ']');
msg := LogMsg (msg);
*)
54 : DIST(COND:=COND,MD0=>MD770,MD1=>MD771,MD2=>MD772,MD3=>MD773,MD4=>MD774);
55 : DIST(COND:=COND,MD0=>MD775,MD1=>MD776,MD2=>MD777,MD3=>MD778,MD4=>MD779);
56 : DIST(COND:=COND,MD0=>MD780,MD1=>MD781,MD2=>MD782,MD3=>MD783,MD4=>MD784);
57 : DIST(COND:=COND,MD0=>MD785,MD1=>MD786,MD2=>MD787,MD3=>MD788,MD4=>MD789);
58 : DIST(COND:=COND,MD0=>MD790,MD1=>MD791,MD2=>MD792,MD3=>MD793,MD4=>MD794);
59 : DIST(COND:=COND,MD0=>MD795,MD1=>MD796,MD2=>MD797,MD3=>MD798,MD4=>MD799);

60 : DIST(COND:=COND,MD0=>MD800,MD1=>MD801,MD2=>MD802,MD3=>MD803,MD4=>MD804);
61 : DIST(COND:=COND,MD0=>MD805,MD1=>MD806,MD2=>MD807,MD3=>MD808,MD4=>MD809);
62 : DIST(COND:=COND,MD0=>MD810,MD1=>MD811,MD2=>MD812,MD3=>MD813,MD4=>MD814);
63 : DIST(COND:=COND,MD0=>MD815,MD1=>MD816,MD2=>MD817,MD3=>MD818,MD4=>MD819);
64 : DIST(COND:=COND,MD0=>MD820,MD1=>MD821,MD2=>MD822,MD3=>MD823,MD4=>MD824);
65 : DIST(COND:=COND,MD0=>MD825,MD1=>MD826,MD2=>MD827,MD3=>MD828,MD4=>MD829);
66 : DIST(COND:=COND,MD0=>MD830,MD1=>MD831,MD2=>MD832,MD3=>MD833,MD4=>MD834);
67 : DIST(COND:=COND,MD0=>MD835,MD1=>MD836,MD2=>MD837,MD3=>MD838,MD4=>MD839);
68 : DIST(COND:=COND,MD0=>MD840,MD1=>MD841,MD2=>MD842,MD3=>MD843,MD4=>MD844);
69 : DIST(COND:=COND,MD0=>MD845,MD1=>MD846,MD2=>MD847,MD3=>MD848,MD4=>MD849);

